// TwinCAT 3 PLC project PLC
// ProgramVersion: 3.1.4023.0
// libraries:
//   Tc2_Standard, * (Beckhoff Automation GmbH)
//   Tc2_System, * (Beckhoff Automation GmbH)
//   Tc3_Module, * (Beckhoff Automation GmbH)
// project tree:
//   / PlcTask.TcTTO
//   POUs/ MAIN.TcPOU
//   DUTs/IO/PDOs/ InfoData_6F19DB2B.TcDUT, Inputs_CC16D1F4.TcDUT, Outputs_D8BAB3B3.TcDUT, WcState_9091E0EB.TcDUT, InfoData_90184F0C.TcDUT, Channel_954C2EED.TcDUT, Channel_60E28ED2.TcDUT, Channel_7DE26195.TcDUT, Channel_2E0D480D.TcDUT, Channel_61FC1536.TcDUT, Channel_16463F74.TcDUT, Channel_707BD1FE.TcDUT, Channel_7D202F58.TcDUT, Channel_6CC0E226.TcDUT, Channel_0F0CD940.TcDUT, Channel_87C95E76.TcDUT, Channel_65B76600.TcDUT, Channel_72DF6336.TcDUT, Channel_22DCD695.TcDUT, Channel_3C1A6500.TcDUT, Channel_B5275D8E.TcDUT, Channel_03CEAA5E.TcDUT, Channel_70C997F3.TcDUT, Channel_1D6668A9.TcDUT, Channel_6B723A16.TcDUT, Channel_460B8C40.TcDUT, Channel_DCF170BB.TcDUT, Channel_26FC8FD8.TcDUT, Channel_FEA3DBF8.TcDUT, Channel_0D1929F0.TcDUT, Channel_6576A681.TcDUT, Channel_2589C8DC.TcDUT, Channel_BF3661CD.TcDUT, Channel_2EC3E8CA.TcDUT, Channel_F5DB8AD1.TcDUT, Channel_6D8B740B.TcDUT, Channel_2DA3FF3C.TcDUT, Channel_0514A8FA.TcDUT, Channel_4E9D1E2D.TcDUT, Channel_78571FB4.TcDUT, Channel_87905831.TcDUT, Channel_099BCCDA.TcDUT, Channel_82ADD076.TcDUT, Channel_332F026B.TcDUT, Channel_A6A8AB45.TcDUT, Channel_A42BCA5C.TcDUT, Channel_08506BCE.TcDUT, Channel_08533804.TcDUT, Channel_A04AC4BD.TcDUT, Channel_77910383.TcDUT, Channel_9BC0092E.TcDUT, Channel_7606D989.TcDUT, Channel_6931CC5B.TcDUT, Channel_F7FDEFA0.TcDUT, Channel_A1C14FB4.TcDUT, Channel_A4B48F2D.TcDUT, Channel_9E293686.TcDUT, Channel_F84AC14F.TcDUT, Channel_2F314509.TcDUT, Channel_D9D48807.TcDUT, Channel_D13646E3.TcDUT, Channel_3263D8D5.TcDUT, Channel_D490E973.TcDUT, KL_6576A681.TcDUT, Channel_64AAC8C7.TcDUT, Channel_471FAA5C.TcDUT, Diag_1F4F4573.TcDUT, Channel_0029832E.TcDUT, Channel_12652743.TcDUT, InfoData_E68C61CD.TcDUT, WcState_0B2B16F9.TcDUT, InfoData_2A97D6CF.TcDUT, Inputs_25A0042B.TcDUT, Outputs_2397A10E.TcDUT
//   DUTs/IO/Boxes/ EK1100_1FC0878B.TcDUT, BK1250_A2FCADE7.TcDUT, KL_5E2F016F.TcDUT, KL_2EA97E3E.TcDUT, KL_1187B721.TcDUT, KL_E991A364.TcDUT, KL_063F0990.TcDUT, KL_5AE00A1C.TcDUT, KL_CFA8830D.TcDUT, KL_DBC0B844.TcDUT, KL_6930B3B2.TcDUT, KL_4F0DAD84.TcDUT, KL_2227C35B.TcDUT, KL1002_BB38DA8F.TcDUT, KL_E653A8C1.TcDUT, KL1012_BB38DA8F.TcDUT, KL1032_BB38DA8F.TcDUT, KL1052_BB38DA8F.TcDUT, KL1104_4A257D2B.TcDUT, KL1114_4A257D2B.TcDUT, KL1124_4A257D2B.TcDUT, KL1154_4A257D2B.TcDUT, KL1164_4A257D2B.TcDUT, KL1184_4A257D2B.TcDUT, KL1194_4A257D2B.TcDUT, KL1212_EC84F46C.TcDUT, KL1232_BB38DA8F.TcDUT, KL1302_BB38DA8F.TcDUT, KL1304_4A257D2B.TcDUT, KL1312_BB38DA8F.TcDUT, KL1314_4A257D2B.TcDUT, KL1352_B54AC54D.TcDUT, KL1362_B54AC54D.TcDUT, KL1382_B54AC54D.TcDUT, KL1402_BB38DA8F.TcDUT, KL1404_4A257D2B.TcDUT, KL1408_8EF4D3E9.TcDUT, KL1412_BB38DA8F.TcDUT, KL1414_4A257D2B.TcDUT, KL1418_8EF4D3E9.TcDUT, KL1434_4A257D2B.TcDUT, KL1488_8EF4D3E9.TcDUT, KL1498_8EF4D3E9.TcDUT, KL1501_EE1D4506.TcDUT, KL_62DC61BC.TcDUT, KL1512_78388DBB.TcDUT, KL1702_BB38DA8F.TcDUT, KL1704_4A257D2B.TcDUT, KL1712_BB38DA8F.TcDUT, KL_BB38DA8F.TcDUT, KL1722_BB38DA8F.TcDUT, KL1804_4A257D2B.TcDUT, KL1808_8EF4D3E9.TcDUT, KL1809_65B88BEE.TcDUT, KL1814_4A257D2B.TcDUT, KL1819_65B88BEE.TcDUT, KL1859_C5B2A062.TcDUT, KL1862_65B88BEE.TcDUT, KL_65B88BEE.TcDUT, KL1872_65B88BEE.TcDUT, KL1889_65B88BEE.TcDUT, KL1904_7F0D69A9.TcDUT, KL1908_7F0D69A9.TcDUT, KL_ABE34026.TcDUT, KL_E882B8F1.TcDUT, KL_52751275.TcDUT, KL2012_DCA75612.TcDUT, KL2022_DCA75612.TcDUT, KL2032_DCA75612.TcDUT, KL2114_E49EE1EF.TcDUT, KL2124_E49EE1EF.TcDUT, KL2134_E49EE1EF.TcDUT, KL2184_E49EE1EF.TcDUT, KL2212_BA18203A.TcDUT, KL1202_EC84F46C.TcDUT, KL2404_E49EE1EF.TcDUT, KL2408_CBAD53BF.TcDUT, KL2424_E49EE1EF.TcDUT, KL2442_DCA75612.TcDUT, KL2488_CBAD53BF.TcDUT, KL2284_008A18FD.TcDUT, KL2502_78388DBB.TcDUT, KL2512_78388DBB.TcDUT, KL2521_D5F34107.TcDUT, KL2531_D5AE5504.TcDUT, KL_5C335388.TcDUT, KL2532_B0461874.TcDUT, KL2535_B0461874.TcDUT, KL_501418F2.TcDUT, KL2541_D5AE5504.TcDUT, KL2542_B0461874.TcDUT, KL2545_B0461874.TcDUT, KL2552_B0461874.TcDUT, KL2602_DCA75612.TcDUT, KL_DCA75612.TcDUT, KL2612_DCA75612.TcDUT, KL2622_DCA75612.TcDUT, KL2631_DE78D366.TcDUT, KL2634_E49EE1EF.TcDUT, KL2641_8487B205.TcDUT, KL_AF699C3C.TcDUT, KL2652_DCA75612.TcDUT, KL_6148C904.TcDUT, KL2701_DE78D366.TcDUT, KL2702_DCA75612.TcDUT, KL2712_DCA75612.TcDUT, KL2722_DCA75612.TcDUT, KL2732_DCA75612.TcDUT, KL2744_E49EE1EF.TcDUT, KL2751_6148C904.TcDUT, KL2761_6148C904.TcDUT, KL2784_E49EE1EF.TcDUT, KL2791_6148C904.TcDUT, KL2794_E49EE1EF.TcDUT, KL2798_CBAD53BF.TcDUT, KL2808_CBAD53BF.TcDUT, KL2819_28D63841.TcDUT, KL2828_CBAD53BF.TcDUT, KL2809_F0D0C9F8.TcDUT, KL2872_F0D0C9F8.TcDUT, KL2889_F0D0C9F8.TcDUT, KL2904_7F0D69A9.TcDUT, KL_F0D0C9F8.TcDUT, KL_CF002DCA.TcDUT, KL_F7A5EEBF.TcDUT, KL_E49EE1EF.TcDUT, KL_F206FFFF.TcDUT, KL_13ED1AE5.TcDUT, KL2774_6148C904.TcDUT, KL_CBAD53BF.TcDUT, KL3001_6148C904.TcDUT, KL3002_B0461874.TcDUT, KL3011_6148C904.TcDUT, KL3012_B0461874.TcDUT, KL3021_6148C904.TcDUT, KL3022_B0461874.TcDUT, KL3041_6148C904.TcDUT, KL3042_B0461874.TcDUT, KL3044_8BE38B75.TcDUT, KL_ACD69469.TcDUT, KL3051_6148C904.TcDUT, KL3052_B0461874.TcDUT, KL3054_8BE38B75.TcDUT, KL3061_6148C904.TcDUT, KL3062_B0461874.TcDUT, KL3064_8BE38B75.TcDUT, KL3102_B0461874.TcDUT, KL3112_B0461874.TcDUT, KL3122_B0461874.TcDUT, KL3132_B0461874.TcDUT, KL3142_78388DBB.TcDUT, KL3152_78388DBB.TcDUT, KL3158_8BE38B75.TcDUT, KL3162_78388DBB.TcDUT, KL3172_78388DBB.TcDUT, KL_78388DBB.TcDUT, KL3182_B0461874.TcDUT, KL3201_6148C904.TcDUT, KL3202_B0461874.TcDUT, KL3204_8BE38B75.TcDUT, KL_8BE38B75.TcDUT, KL3214_8BE38B75.TcDUT, KL3222_B0461874.TcDUT, KL3224_8BE38B75.TcDUT, KL3228_8BE38B75.TcDUT, KL3302_B0461874.TcDUT, KL3311_6148C904.TcDUT, KL3312_B0461874.TcDUT, KL3314_8BE38B75.TcDUT, KL3351_33637CB0.TcDUT, KL_C7B8B3CA.TcDUT, KL3356_E004D4E2.TcDUT, KL_EE1D4506.TcDUT, KL3361_73CB82BA.TcDUT, KL_73CB82BA.TcDUT, KL3362_E98BF8F1.TcDUT, KL6211_60136EA1.TcDUT, KL_9AE543B6.TcDUT, KL_FC0201B8.TcDUT, KL_498D8863.TcDUT, KL_71341691.TcDUT, KL_2B11657C.TcDUT, KL6224_C0F107BD.TcDUT, KL_FC1E3393.TcDUT, KL_C51B1CB0.TcDUT, KL_7EC2CD64.TcDUT, KL_3829421A.TcDUT, KL_9116C2C1.TcDUT, KL6551_528AE398.TcDUT, KL_3325E583.TcDUT, KL_528AE398.TcDUT, KL6781_BE595CA2.TcDUT, KL6811_6148C904.TcDUT, KL6821_F77C82D2.TcDUT, KL6831_BE595CA2.TcDUT, KL6841_BE595CA2.TcDUT, KL6904_B938D612.TcDUT, KL_921B772D.TcDUT, KL_779990DF.TcDUT, KL8001_7761653A.TcDUT, KL8519_8C34650F.TcDUT, KL8524_A4B9216E.TcDUT, KL8528_73A97EC1.TcDUT, KL8548_23451728.TcDUT, KL8610_C571D068.TcDUT, KL_5A83E84C.TcDUT, KL_BF4AA06C.TcDUT, KL_7485E925.TcDUT, KL_372C6BEC.TcDUT, KL_2E5CD6C8.TcDUT, KL_68BDE1E9.TcDUT, KL_84AAE8B6.TcDUT, KL9110_8BEE55F2.TcDUT, KL9160_8BEE55F2.TcDUT, KL9191_962A24DF.TcDUT, KL9210_8BEE55F2.TcDUT, KL9260_8BEE55F2.TcDUT, KL_E4BD2B38.TcDUT, KL9528_8C984603.TcDUT, KL9999_7A10A7F6.TcDUT
//   DUTs/IO/Devices/ SyncUnitTask_2D604ED5.TcDUT, SyncUnitTasks_6FEB8257.TcDUT, SyncUnits_99E584AF.TcDUT
//   DUTs/IO/Topology/ TcTerminals210_1BK1250_A7ABB5AA.TcDUT, TcTerminals210_1EK1100_5C778379.TcDUT, TcTerminals210_2BK1250_CEF74155.TcDUT, TcTerminals210_2EK1100_50C14331.TcDUT, EtherCAT_Master_KL_4053F38C.TcDUT, EtherCAT_Master_KL_8A657514.TcDUT, EtherCAT_Master_KL_B156B97E.TcDUT
//   DUTs/IO/Base/ EtcSlaveBase_82538BE2.TcDUT, EtcSlaveBase_82538BE2.TcDUT, EtcSlaveBase_82538BE2.TcDUT, EtcSlaveTerminalBase_947E5A46.TcDUT, EtcSlaveBoxBase_77A0E4A7.TcDUT, EtcSlaveEndTerminalBase_866C7F0C.TcDUT, InputBase_8311D824.TcDUT, OutputBase_10CEE7DE.TcDUT, EtcMasterBase_62654B43.TcDUT
//   GVLs/ GVL_iXlinker.TcGVL

CONFIGURATION PLC
    RESOURCE PLC ON TwinCAT3
        TASK PlcTask(INTERVAL := T#10ms, PRIORITY := 20);
        PROGRAM MAIN WITH PlcTask : MAIN;
    END_RESOURCE
END_CONFIGURATION

// ---- DUTs/IO/PDOs/InfoData_6F19DB2B.TcDUT
{attribute 'GeneratedUsingTerminal: EK1100-0000-0018'}
{attribute addProperty BoxType "EK1100-0000-0018"}
{attribute addProperty Id "StateAT %I*UINT2"}
{attribute addProperty CRC "1863965483"}
{attribute addProperty Size "2"}
TYPE InfoData_6F19DB2B :
STRUCT
	{attribute addProperty Name "State"}
	State AT %I* : UINT;
END_STRUCT
END_TYPE

// ---- DUTs/IO/PDOs/Inputs_CC16D1F4.TcDUT
{attribute 'GeneratedUsingTerminal: BK1250-0000-0019'}
{attribute addProperty BoxType "BK1250-0000-0019"}
{attribute addProperty Id "CouplerStateAT %I*UINT0"}
{attribute addProperty CRC "3424047604"}
{attribute addProperty Size "0"}
TYPE Inputs_CC16D1F4 EXTENDS InputBase_8311D824 :
STRUCT
	{attribute addProperty Name "CouplerState"}
	CouplerState AT %I* : UINT;
END_STRUCT
END_TYPE

// ---- DUTs/IO/PDOs/Outputs_D8BAB3B3.TcDUT
{attribute 'GeneratedUsingTerminal: BK1250-0000-0019'}
{attribute addProperty BoxType "BK1250-0000-0019"}
{attribute addProperty Id "CouplerCtrlAT %I*UINT0"}
{attribute addProperty CRC "3636114355"}
{attribute addProperty Size "0"}
TYPE Outputs_D8BAB3B3 EXTENDS InputBase_8311D824 :
STRUCT
	{attribute addProperty Name "CouplerCtrl"}
	CouplerCtrl AT %I* : UINT;
END_STRUCT
END_TYPE

// ---- DUTs/IO/PDOs/WcState_9091E0EB.TcDUT
{attribute 'GeneratedUsingTerminal: BK1250-0000-0019'}
{attribute addProperty BoxType "BK1250-0000-0019"}
{attribute addProperty Id "WcStateAT %I*BOOL1InputToggleAT %I*BOOL1"}
{attribute addProperty CRC "2425479403"}
{attribute addProperty Size "2"}
TYPE WcState_9091E0EB :
STRUCT
	{attribute addProperty Name "WcState"}
	WcState AT %I* : BOOL;
	{attribute addProperty Name "InputToggle"}
	InputToggle AT %I* : BOOL;
END_STRUCT
END_TYPE

// ---- DUTs/IO/PDOs/InfoData_90184F0C.TcDUT
{attribute 'GeneratedUsingTerminal: BK1250-0000-0019'}
{attribute addProperty BoxType "BK1250-0000-0019"}
{attribute addProperty Id "AdsAddrAT %I*AMSADDR8AoeNetIdAT %I*AMSNETID6StateAT %I*UINT2"}
{attribute addProperty CRC "2417512204"}
{attribute addProperty Size "16"}
TYPE InfoData_90184F0C EXTENDS InputBase_8311D824 :
STRUCT
	{attribute addProperty Name "AdsAddr"}
	AdsAddr AT %I* : AMSADDR;
	{attribute addProperty Name "AoeNetId"}
	AoeNetId AT %I* : AMSNETID;
	{attribute addProperty Name "State"}
	State AT %I* : UINT;
END_STRUCT
END_TYPE

// ---- DUTs/IO/PDOs/Channel_954C2EED.TcDUT
{attribute 'GeneratedUsingTerminal: KL9940-0050'}
{attribute addProperty BoxType "KL9940-0050"}
{attribute addProperty Id "Key_1AT %I*BOOL0Key_2AT %I*BOOL0Key_3AT %I*BOOL0Key_4AT %I*BOOL0Key_5AT %I*BOOL0Key_6AT %I*BOOL0Key_7AT %I*BOOL0Key_8AT %I*BOOL0Key_9AT %I*BOOL0Key_10AT %I*BOOL0Key_11AT %I*BOOL0Key_12AT %I*BOOL0Key_13AT %I*BOOL0Key_14AT %I*BOOL0Key_15AT %I*BOOL0Key_16AT %I*BOOL0Key_17AT %I*BOOL0Key_18AT %I*BOOL0Key_19AT %I*BOOL0Key_20AT %I*BOOL0Key_21AT %I*BOOL0Key_22AT %I*BOOL0Key_23AT %I*BOOL0Key_24AT %I*BOOL0Key_25AT %I*BOOL0Key_26AT %I*BOOL0Key_27AT %I*BOOL0Key_28AT %I*BOOL0Key_29AT %I*BOOL0Key_30AT %I*BOOL0Key_31AT %I*BOOL0Key_32AT %I*BOOL0Key_33AT %I*BOOL0Key_34AT %I*BOOL0Key_35AT %I*BOOL0Key_36AT %I*BOOL0Key_37AT %I*BOOL0Key_38AT %I*BOOL0Key_39AT %I*BOOL0Key_40AT %I*BOOL0"}
{attribute addProperty CRC "2504797933"}
{attribute addProperty Size "0"}
TYPE Channel_954C2EED EXTENDS InputBase_8311D824 :
STRUCT
	{attribute addProperty Name "Key_1"}
	Key_1 AT %I* : BOOL;
	{attribute addProperty Name "Key_2"}
	Key_2 AT %I* : BOOL;
	{attribute addProperty Name "Key_3"}
	Key_3 AT %I* : BOOL;
	{attribute addProperty Name "Key_4"}
	Key_4 AT %I* : BOOL;
	{attribute addProperty Name "Key_5"}
	Key_5 AT %I* : BOOL;
	{attribute addProperty Name "Key_6"}
	Key_6 AT %I* : BOOL;
	{attribute addProperty Name "Key_7"}
	Key_7 AT %I* : BOOL;
	{attribute addProperty Name "Key_8"}
	Key_8 AT %I* : BOOL;
	{attribute addProperty Name "Key_9"}
	Key_9 AT %I* : BOOL;
	{attribute addProperty Name "Key_10"}
	Key_10 AT %I* : BOOL;
	{attribute addProperty Name "Key_11"}
	Key_11 AT %I* : BOOL;
	{attribute addProperty Name "Key_12"}
	Key_12 AT %I* : BOOL;
	{attribute addProperty Name "Key_13"}
	Key_13 AT %I* : BOOL;
	{attribute addProperty Name "Key_14"}
	Key_14 AT %I* : BOOL;
	{attribute addProperty Name "Key_15"}
	Key_15 AT %I* : BOOL;
	{attribute addProperty Name "Key_16"}
	Key_16 AT %I* : BOOL;
	{attribute addProperty Name "Key_17"}
	Key_17 AT %I* : BOOL;
	{attribute addProperty Name "Key_18"}
	Key_18 AT %I* : BOOL;
	{attribute addProperty Name "Key_19"}
	Key_19 AT %I* : BOOL;
	{attribute addProperty Name "Key_20"}
	Key_20 AT %I* : BOOL;
	{attribute addProperty Name "Key_21"}
	Key_21 AT %I* : BOOL;
	{attribute addProperty Name "Key_22"}
	Key_22 AT %I* : BOOL;
	{attribute addProperty Name "Key_23"}
	Key_23 AT %I* : BOOL;
	{attribute addProperty Name "Key_24"}
	Key_24 AT %I* : BOOL;
	{attribute addProperty Name "Key_25"}
	Key_25 AT %I* : BOOL;
	{attribute addProperty Name "Key_26"}
	Key_26 AT %I* : BOOL;
	{attribute addProperty Name "Key_27"}
	Key_27 AT %I* : BOOL;
	{attribute addProperty Name "Key_28"}
	Key_28 AT %I* : BOOL;
	{attribute addProperty Name "Key_29"}
	Key_29 AT %I* : BOOL;
	{attribute addProperty Name "Key_30"}
	Key_30 AT %I* : BOOL;
	{attribute addProperty Name "Key_31"}
	Key_31 AT %I* : BOOL;
	{attribute addProperty Name "Key_32"}
	Key_32 AT %I* : BOOL;
	{attribute addProperty Name "Key_33"}
	Key_33 AT %I* : BOOL;
	{attribute addProperty Name "Key_34"}
	Key_34 AT %I* : BOOL;
	{attribute addProperty Name "Key_35"}
	Key_35 AT %I* : BOOL;
	{attribute addProperty Name "Key_36"}
	Key_36 AT %I* : BOOL;
	{attribute addProperty Name "Key_37"}
	Key_37 AT %I* : BOOL;
	{attribute addProperty Name "Key_38"}
	Key_38 AT %I* : BOOL;
	{attribute addProperty Name "Key_39"}
	Key_39 AT %I* : BOOL;
	{attribute addProperty Name "Key_40"}
	Key_40 AT %I* : BOOL;
END_STRUCT
END_TYPE

// ---- DUTs/IO/PDOs/Channel_60E28ED2.TcDUT
{attribute 'GeneratedUsingTerminal: KL9900-0054'}
{attribute addProperty BoxType "KL9900-0054"}
{attribute addProperty Id "Key_1AT %I*BOOL0Key_2AT %I*BOOL0Key_3AT %I*BOOL0Key_4AT %I*BOOL0LED_1AT %Q*BOOL0LED_2AT %Q*BOOL0LED_3AT %Q*BOOL0LED_4AT %Q*BOOL0"}
{attribute addProperty CRC "1625460434"}
{attribute addProperty Size "0"}
TYPE Channel_60E28ED2 :
STRUCT
	{attribute addProperty Name "Key_1"}
	Key_1 AT %I* : BOOL;
	{attribute addProperty Name "Key_2"}
	Key_2 AT %I* : BOOL;
	{attribute addProperty Name "Key_3"}
	Key_3 AT %I* : BOOL;
	{attribute addProperty Name "Key_4"}
	Key_4 AT %I* : BOOL;
	{attribute addProperty Name "LED_1"}
	LED_1 AT %Q* : BOOL;
	{attribute addProperty Name "LED_2"}
	LED_2 AT %Q* : BOOL;
	{attribute addProperty Name "LED_3"}
	LED_3 AT %Q* : BOOL;
	{attribute addProperty Name "LED_4"}
	LED_4 AT %Q* : BOOL;
END_STRUCT
END_TYPE

// ---- DUTs/IO/PDOs/Channel_7DE26195.TcDUT
{attribute 'GeneratedUsingTerminal: KL9900-0055'}
{attribute addProperty BoxType "KL9900-0055"}
{attribute addProperty Id "Key_1AT %I*BOOL0Key_2AT %I*BOOL0Key_3AT %I*BOOL0Key_4AT %I*BOOL0Key_5AT %I*BOOL0Key_6AT %I*BOOL0Key_7AT %I*BOOL0Key_8AT %I*BOOL0LED_1AT %Q*BOOL0LED_2AT %Q*BOOL0LED_3AT %Q*BOOL0LED_4AT %Q*BOOL0LED_5AT %Q*BOOL0LED_6AT %Q*BOOL0LED_7AT %Q*BOOL0LED_8AT %Q*BOOL0"}
{attribute addProperty CRC "2111988117"}
{attribute addProperty Size "0"}
TYPE Channel_7DE26195 :
STRUCT
	{attribute addProperty Name "Key_1"}
	Key_1 AT %I* : BOOL;
	{attribute addProperty Name "Key_2"}
	Key_2 AT %I* : BOOL;
	{attribute addProperty Name "Key_3"}
	Key_3 AT %I* : BOOL;
	{attribute addProperty Name "Key_4"}
	Key_4 AT %I* : BOOL;
	{attribute addProperty Name "Key_5"}
	Key_5 AT %I* : BOOL;
	{attribute addProperty Name "Key_6"}
	Key_6 AT %I* : BOOL;
	{attribute addProperty Name "Key_7"}
	Key_7 AT %I* : BOOL;
	{attribute addProperty Name "Key_8"}
	Key_8 AT %I* : BOOL;
	{attribute addProperty Name "LED_1"}
	LED_1 AT %Q* : BOOL;
	{attribute addProperty Name "LED_2"}
	LED_2 AT %Q* : BOOL;
	{attribute addProperty Name "LED_3"}
	LED_3 AT %Q* : BOOL;
	{attribute addProperty Name "LED_4"}
	LED_4 AT %Q* : BOOL;
	{attribute addProperty Name "LED_5"}
	LED_5 AT %Q* : BOOL;
	{attribute addProperty Name "LED_6"}
	LED_6 AT %Q* : BOOL;
	{attribute addProperty Name "LED_7"}
	LED_7 AT %Q* : BOOL;
	{attribute addProperty Name "LED_8"}
	LED_8 AT %Q* : BOOL;
END_STRUCT
END_TYPE

// ---- DUTs/IO/PDOs/Channel_2E0D480D.TcDUT
{attribute 'GeneratedUsingTerminal: KL9900-0056'}
{attribute addProperty BoxType "KL9900-0056"}
{attribute addProperty Id "Key_1AT %I*BOOL0Key_2AT %I*BOOL0Key_3AT %I*BOOL0Key_4AT %I*BOOL0Key_5AT %I*BOOL0Key_6AT %I*BOOL0Key_7AT %I*BOOL0Key_8AT %I*BOOL0Key_9AT %I*BOOL0Key_10AT %I*BOOL0Key_11AT %I*BOOL0Key_12AT %I*BOOL0LED_1AT %Q*BOOL0LED_2AT %Q*BOOL0LED_3AT %Q*BOOL0LED_4AT %Q*BOOL0LED_5AT %Q*BOOL0LED_6AT %Q*BOOL0LED_7AT %Q*BOOL0LED_8AT %Q*BOOL0LED_9AT %Q*BOOL0LED_10AT %Q*BOOL0LED_11AT %Q*BOOL0LED_12AT %Q*BOOL0"}
{attribute addProperty CRC "772622349"}
{attribute addProperty Size "0"}
TYPE Channel_2E0D480D :
STRUCT
	{attribute addProperty Name "Key_1"}
	Key_1 AT %I* : BOOL;
	{attribute addProperty Name "Key_2"}
	Key_2 AT %I* : BOOL;
	{attribute addProperty Name "Key_3"}
	Key_3 AT %I* : BOOL;
	{attribute addProperty Name "Key_4"}
	Key_4 AT %I* : BOOL;
	{attribute addProperty Name "Key_5"}
	Key_5 AT %I* : BOOL;
	{attribute addProperty Name "Key_6"}
	Key_6 AT %I* : BOOL;
	{attribute addProperty Name "Key_7"}
	Key_7 AT %I* : BOOL;
	{attribute addProperty Name "Key_8"}
	Key_8 AT %I* : BOOL;
	{attribute addProperty Name "Key_9"}
	Key_9 AT %I* : BOOL;
	{attribute addProperty Name "Key_10"}
	Key_10 AT %I* : BOOL;
	{attribute addProperty Name "Key_11"}
	Key_11 AT %I* : BOOL;
	{attribute addProperty Name "Key_12"}
	Key_12 AT %I* : BOOL;
	{attribute addProperty Name "LED_1"}
	LED_1 AT %Q* : BOOL;
	{attribute addProperty Name "LED_2"}
	LED_2 AT %Q* : BOOL;
	{attribute addProperty Name "LED_3"}
	LED_3 AT %Q* : BOOL;
	{attribute addProperty Name "LED_4"}
	LED_4 AT %Q* : BOOL;
	{attribute addProperty Name "LED_5"}
	LED_5 AT %Q* : BOOL;
	{attribute addProperty Name "LED_6"}
	LED_6 AT %Q* : BOOL;
	{attribute addProperty Name "LED_7"}
	LED_7 AT %Q* : BOOL;
	{attribute addProperty Name "LED_8"}
	LED_8 AT %Q* : BOOL;
	{attribute addProperty Name "LED_9"}
	LED_9 AT %Q* : BOOL;
	{attribute addProperty Name "LED_10"}
	LED_10 AT %Q* : BOOL;
	{attribute addProperty Name "LED_11"}
	LED_11 AT %Q* : BOOL;
	{attribute addProperty Name "LED_12"}
	LED_12 AT %Q* : BOOL;
END_STRUCT
END_TYPE

// ---- DUTs/IO/PDOs/Channel_61FC1536.TcDUT
{attribute 'GeneratedUsingTerminal: KL9900-0057'}
{attribute addProperty BoxType "KL9900-0057"}
{attribute addProperty Id "Key_1AT %I*BOOL0Key_2AT %I*BOOL0Key_3AT %I*BOOL0Key_4AT %I*BOOL0Key_5AT %I*BOOL0Key_6AT %I*BOOL0Key_7AT %I*BOOL0Key_8AT %I*BOOL0Key_9AT %I*BOOL0Key_10AT %I*BOOL0Key_11AT %I*BOOL0Key_12AT %I*BOOL0Key_13AT %I*BOOL0Key_14AT %I*BOOL0Key_15AT %I*BOOL0Key_16AT %I*BOOL0LED_1AT %Q*BOOL0LED_2AT %Q*BOOL0LED_3AT %Q*BOOL0LED_4AT %Q*BOOL0LED_5AT %Q*BOOL0LED_6AT %Q*BOOL0LED_7AT %Q*BOOL0LED_8AT %Q*BOOL0LED_9AT %Q*BOOL0LED_10AT %Q*BOOL0LED_11AT %Q*BOOL0LED_12AT %Q*BOOL0LED_13AT %Q*BOOL0LED_14AT %Q*BOOL0LED_15AT %Q*BOOL0LED_16AT %Q*BOOL0"}
{attribute addProperty CRC "1643910454"}
{attribute addProperty Size "0"}
TYPE Channel_61FC1536 :
STRUCT
	{attribute addProperty Name "Key_1"}
	Key_1 AT %I* : BOOL;
	{attribute addProperty Name "Key_2"}
	Key_2 AT %I* : BOOL;
	{attribute addProperty Name "Key_3"}
	Key_3 AT %I* : BOOL;
	{attribute addProperty Name "Key_4"}
	Key_4 AT %I* : BOOL;
	{attribute addProperty Name "Key_5"}
	Key_5 AT %I* : BOOL;
	{attribute addProperty Name "Key_6"}
	Key_6 AT %I* : BOOL;
	{attribute addProperty Name "Key_7"}
	Key_7 AT %I* : BOOL;
	{attribute addProperty Name "Key_8"}
	Key_8 AT %I* : BOOL;
	{attribute addProperty Name "Key_9"}
	Key_9 AT %I* : BOOL;
	{attribute addProperty Name "Key_10"}
	Key_10 AT %I* : BOOL;
	{attribute addProperty Name "Key_11"}
	Key_11 AT %I* : BOOL;
	{attribute addProperty Name "Key_12"}
	Key_12 AT %I* : BOOL;
	{attribute addProperty Name "Key_13"}
	Key_13 AT %I* : BOOL;
	{attribute addProperty Name "Key_14"}
	Key_14 AT %I* : BOOL;
	{attribute addProperty Name "Key_15"}
	Key_15 AT %I* : BOOL;
	{attribute addProperty Name "Key_16"}
	Key_16 AT %I* : BOOL;
	{attribute addProperty Name "LED_1"}
	LED_1 AT %Q* : BOOL;
	{attribute addProperty Name "LED_2"}
	LED_2 AT %Q* : BOOL;
	{attribute addProperty Name "LED_3"}
	LED_3 AT %Q* : BOOL;
	{attribute addProperty Name "LED_4"}
	LED_4 AT %Q* : BOOL;
	{attribute addProperty Name "LED_5"}
	LED_5 AT %Q* : BOOL;
	{attribute addProperty Name "LED_6"}
	LED_6 AT %Q* : BOOL;
	{attribute addProperty Name "LED_7"}
	LED_7 AT %Q* : BOOL;
	{attribute addProperty Name "LED_8"}
	LED_8 AT %Q* : BOOL;
	{attribute addProperty Name "LED_9"}
	LED_9 AT %Q* : BOOL;
	{attribute addProperty Name "LED_10"}
	LED_10 AT %Q* : BOOL;
	{attribute addProperty Name "LED_11"}
	LED_11 AT %Q* : BOOL;
	{attribute addProperty Name "LED_12"}
	LED_12 AT %Q* : BOOL;
	{attribute addProperty Name "LED_13"}
	LED_13 AT %Q* : BOOL;
	{attribute addProperty Name "LED_14"}
	LED_14 AT %Q* : BOOL;
	{attribute addProperty Name "LED_15"}
	LED_15 AT %Q* : BOOL;
	{attribute addProperty Name "LED_16"}
	LED_16 AT %Q* : BOOL;
END_STRUCT
END_TYPE

// ---- DUTs/IO/PDOs/Channel_16463F74.TcDUT
{attribute 'GeneratedUsingTerminal: KL9900-0058'}
{attribute addProperty BoxType "KL9900-0058"}
{attribute addProperty Id "Key_1AT %I*BOOL0Key_2AT %I*BOOL0Key_3AT %I*BOOL0Key_4AT %I*BOOL0Key_5AT %I*BOOL0Key_6AT %I*BOOL0Key_7AT %I*BOOL0Key_8AT %I*BOOL0Key_9AT %I*BOOL0Key_10AT %I*BOOL0Key_11AT %I*BOOL0Key_12AT %I*BOOL0Key_13AT %I*BOOL0Key_14AT %I*BOOL0Key_15AT %I*BOOL0Key_16AT %I*BOOL0Key_17AT %I*BOOL0Key_18AT %I*BOOL0Key_19AT %I*BOOL0Key_20AT %I*BOOL0LED_1AT %Q*BOOL0LED_2AT %Q*BOOL0LED_3AT %Q*BOOL0LED_4AT %Q*BOOL0LED_5AT %Q*BOOL0LED_6AT %Q*BOOL0LED_7AT %Q*BOOL0LED_8AT %Q*BOOL0LED_9AT %Q*BOOL0LED_10AT %Q*BOOL0LED_11AT %Q*BOOL0LED_12AT %Q*BOOL0LED_13AT %Q*BOOL0LED_14AT %Q*BOOL0LED_15AT %Q*BOOL0LED_16AT %Q*BOOL0LED_17AT %Q*BOOL0LED_18AT %Q*BOOL0LED_19AT %Q*BOOL0LED_20AT %Q*BOOL0"}
{attribute addProperty CRC "373702516"}
{attribute addProperty Size "0"}
TYPE Channel_16463F74 :
STRUCT
	{attribute addProperty Name "Key_1"}
	Key_1 AT %I* : BOOL;
	{attribute addProperty Name "Key_2"}
	Key_2 AT %I* : BOOL;
	{attribute addProperty Name "Key_3"}
	Key_3 AT %I* : BOOL;
	{attribute addProperty Name "Key_4"}
	Key_4 AT %I* : BOOL;
	{attribute addProperty Name "Key_5"}
	Key_5 AT %I* : BOOL;
	{attribute addProperty Name "Key_6"}
	Key_6 AT %I* : BOOL;
	{attribute addProperty Name "Key_7"}
	Key_7 AT %I* : BOOL;
	{attribute addProperty Name "Key_8"}
	Key_8 AT %I* : BOOL;
	{attribute addProperty Name "Key_9"}
	Key_9 AT %I* : BOOL;
	{attribute addProperty Name "Key_10"}
	Key_10 AT %I* : BOOL;
	{attribute addProperty Name "Key_11"}
	Key_11 AT %I* : BOOL;
	{attribute addProperty Name "Key_12"}
	Key_12 AT %I* : BOOL;
	{attribute addProperty Name "Key_13"}
	Key_13 AT %I* : BOOL;
	{attribute addProperty Name "Key_14"}
	Key_14 AT %I* : BOOL;
	{attribute addProperty Name "Key_15"}
	Key_15 AT %I* : BOOL;
	{attribute addProperty Name "Key_16"}
	Key_16 AT %I* : BOOL;
	{attribute addProperty Name "Key_17"}
	Key_17 AT %I* : BOOL;
	{attribute addProperty Name "Key_18"}
	Key_18 AT %I* : BOOL;
	{attribute addProperty Name "Key_19"}
	Key_19 AT %I* : BOOL;
	{attribute addProperty Name "Key_20"}
	Key_20 AT %I* : BOOL;
	{attribute addProperty Name "LED_1"}
	LED_1 AT %Q* : BOOL;
	{attribute addProperty Name "LED_2"}
	LED_2 AT %Q* : BOOL;
	{attribute addProperty Name "LED_3"}
	LED_3 AT %Q* : BOOL;
	{attribute addProperty Name "LED_4"}
	LED_4 AT %Q* : BOOL;
	{attribute addProperty Name "LED_5"}
	LED_5 AT %Q* : BOOL;
	{attribute addProperty Name "LED_6"}
	LED_6 AT %Q* : BOOL;
	{attribute addProperty Name "LED_7"}
	LED_7 AT %Q* : BOOL;
	{attribute addProperty Name "LED_8"}
	LED_8 AT %Q* : BOOL;
	{attribute addProperty Name "LED_9"}
	LED_9 AT %Q* : BOOL;
	{attribute addProperty Name "LED_10"}
	LED_10 AT %Q* : BOOL;
	{attribute addProperty Name "LED_11"}
	LED_11 AT %Q* : BOOL;
	{attribute addProperty Name "LED_12"}
	LED_12 AT %Q* : BOOL;
	{attribute addProperty Name "LED_13"}
	LED_13 AT %Q* : BOOL;
	{attribute addProperty Name "LED_14"}
	LED_14 AT %Q* : BOOL;
	{attribute addProperty Name "LED_15"}
	LED_15 AT %Q* : BOOL;
	{attribute addProperty Name "LED_16"}
	LED_16 AT %Q* : BOOL;
	{attribute addProperty Name "LED_17"}
	LED_17 AT %Q* : BOOL;
	{attribute addProperty Name "LED_18"}
	LED_18 AT %Q* : BOOL;
	{attribute addProperty Name "LED_19"}
	LED_19 AT %Q* : BOOL;
	{attribute addProperty Name "LED_20"}
	LED_20 AT %Q* : BOOL;
END_STRUCT
END_TYPE

// ---- DUTs/IO/PDOs/Channel_707BD1FE.TcDUT
{attribute 'GeneratedUsingTerminal: KL9900-0059'}
{attribute addProperty BoxType "KL9900-0059"}
{attribute addProperty Id "Key_1AT %I*BOOL0Key_2AT %I*BOOL0Key_3AT %I*BOOL0Key_4AT %I*BOOL0Key_5AT %I*BOOL0Key_6AT %I*BOOL0Key_7AT %I*BOOL0Key_8AT %I*BOOL0Key_9AT %I*BOOL0Key_10AT %I*BOOL0Key_11AT %I*BOOL0Key_12AT %I*BOOL0Key_13AT %I*BOOL0Key_14AT %I*BOOL0Key_15AT %I*BOOL0Key_16AT %I*BOOL0Key_17AT %I*BOOL0Key_18AT %I*BOOL0Key_19AT %I*BOOL0Key_20AT %I*BOOL0Key_21AT %I*BOOL0Key_22AT %I*BOOL0Key_23AT %I*BOOL0Key_24AT %I*BOOL0LED_1AT %Q*BOOL0LED_2AT %Q*BOOL0LED_3AT %Q*BOOL0LED_4AT %Q*BOOL0LED_5AT %Q*BOOL0LED_6AT %Q*BOOL0LED_7AT %Q*BOOL0LED_8AT %Q*BOOL0LED_9AT %Q*BOOL0LED_10AT %Q*BOOL0LED_11AT %Q*BOOL0LED_12AT %Q*BOOL0LED_13AT %Q*BOOL0LED_14AT %Q*BOOL0LED_15AT %Q*BOOL0LED_16AT %Q*BOOL0LED_17AT %Q*BOOL0LED_18AT %Q*BOOL0LED_19AT %Q*BOOL0LED_20AT %Q*BOOL0LED_21AT %Q*BOOL0LED_22AT %Q*BOOL0LED_23AT %Q*BOOL0LED_24AT %Q*BOOL0"}
{attribute addProperty CRC "1887162878"}
{attribute addProperty Size "0"}
TYPE Channel_707BD1FE :
STRUCT
	{attribute addProperty Name "Key_1"}
	Key_1 AT %I* : BOOL;
	{attribute addProperty Name "Key_2"}
	Key_2 AT %I* : BOOL;
	{attribute addProperty Name "Key_3"}
	Key_3 AT %I* : BOOL;
	{attribute addProperty Name "Key_4"}
	Key_4 AT %I* : BOOL;
	{attribute addProperty Name "Key_5"}
	Key_5 AT %I* : BOOL;
	{attribute addProperty Name "Key_6"}
	Key_6 AT %I* : BOOL;
	{attribute addProperty Name "Key_7"}
	Key_7 AT %I* : BOOL;
	{attribute addProperty Name "Key_8"}
	Key_8 AT %I* : BOOL;
	{attribute addProperty Name "Key_9"}
	Key_9 AT %I* : BOOL;
	{attribute addProperty Name "Key_10"}
	Key_10 AT %I* : BOOL;
	{attribute addProperty Name "Key_11"}
	Key_11 AT %I* : BOOL;
	{attribute addProperty Name "Key_12"}
	Key_12 AT %I* : BOOL;
	{attribute addProperty Name "Key_13"}
	Key_13 AT %I* : BOOL;
	{attribute addProperty Name "Key_14"}
	Key_14 AT %I* : BOOL;
	{attribute addProperty Name "Key_15"}
	Key_15 AT %I* : BOOL;
	{attribute addProperty Name "Key_16"}
	Key_16 AT %I* : BOOL;
	{attribute addProperty Name "Key_17"}
	Key_17 AT %I* : BOOL;
	{attribute addProperty Name "Key_18"}
	Key_18 AT %I* : BOOL;
	{attribute addProperty Name "Key_19"}
	Key_19 AT %I* : BOOL;
	{attribute addProperty Name "Key_20"}
	Key_20 AT %I* : BOOL;
	{attribute addProperty Name "Key_21"}
	Key_21 AT %I* : BOOL;
	{attribute addProperty Name "Key_22"}
	Key_22 AT %I* : BOOL;
	{attribute addProperty Name "Key_23"}
	Key_23 AT %I* : BOOL;
	{attribute addProperty Name "Key_24"}
	Key_24 AT %I* : BOOL;
	{attribute addProperty Name "LED_1"}
	LED_1 AT %Q* : BOOL;
	{attribute addProperty Name "LED_2"}
	LED_2 AT %Q* : BOOL;
	{attribute addProperty Name "LED_3"}
	LED_3 AT %Q* : BOOL;
	{attribute addProperty Name "LED_4"}
	LED_4 AT %Q* : BOOL;
	{attribute addProperty Name "LED_5"}
	LED_5 AT %Q* : BOOL;
	{attribute addProperty Name "LED_6"}
	LED_6 AT %Q* : BOOL;
	{attribute addProperty Name "LED_7"}
	LED_7 AT %Q* : BOOL;
	{attribute addProperty Name "LED_8"}
	LED_8 AT %Q* : BOOL;
	{attribute addProperty Name "LED_9"}
	LED_9 AT %Q* : BOOL;
	{attribute addProperty Name "LED_10"}
	LED_10 AT %Q* : BOOL;
	{attribute addProperty Name "LED_11"}
	LED_11 AT %Q* : BOOL;
	{attribute addProperty Name "LED_12"}
	LED_12 AT %Q* : BOOL;
	{attribute addProperty Name "LED_13"}
	LED_13 AT %Q* : BOOL;
	{attribute addProperty Name "LED_14"}
	LED_14 AT %Q* : BOOL;
	{attribute addProperty Name "LED_15"}
	LED_15 AT %Q* : BOOL;
	{attribute addProperty Name "LED_16"}
	LED_16 AT %Q* : BOOL;
	{attribute addProperty Name "LED_17"}
	LED_17 AT %Q* : BOOL;
	{attribute addProperty Name "LED_18"}
	LED_18 AT %Q* : BOOL;
	{attribute addProperty Name "LED_19"}
	LED_19 AT %Q* : BOOL;
	{attribute addProperty Name "LED_20"}
	LED_20 AT %Q* : BOOL;
	{attribute addProperty Name "LED_21"}
	LED_21 AT %Q* : BOOL;
	{attribute addProperty Name "LED_22"}
	LED_22 AT %Q* : BOOL;
	{attribute addProperty Name "LED_23"}
	LED_23 AT %Q* : BOOL;
	{attribute addProperty Name "LED_24"}
	LED_24 AT %Q* : BOOL;
END_STRUCT
END_TYPE

// ---- DUTs/IO/PDOs/Channel_7D202F58.TcDUT
{attribute 'GeneratedUsingTerminal: KL9900-0060'}
{attribute addProperty BoxType "KL9900-0060"}
{attribute addProperty Id "Key_1AT %I*BOOL0Key_2AT %I*BOOL0Key_3AT %I*BOOL0Key_4AT %I*BOOL0Key_5AT %I*BOOL0Key_6AT %I*BOOL0Key_7AT %I*BOOL0Key_8AT %I*BOOL0Key_9AT %I*BOOL0Key_10AT %I*BOOL0Key_11AT %I*BOOL0Key_12AT %I*BOOL0Key_13AT %I*BOOL0Key_14AT %I*BOOL0Key_15AT %I*BOOL0Key_16AT %I*BOOL0Key_17AT %I*BOOL0Key_18AT %I*BOOL0Key_19AT %I*BOOL0Key_20AT %I*BOOL0Key_21AT %I*BOOL0Key_22AT %I*BOOL0Key_23AT %I*BOOL0Key_24AT %I*BOOL0Key_25AT %I*BOOL0Key_26AT %I*BOOL0Key_27AT %I*BOOL0Key_28AT %I*BOOL0LED_1AT %Q*BOOL0LED_2AT %Q*BOOL0LED_3AT %Q*BOOL0LED_4AT %Q*BOOL0LED_5AT %Q*BOOL0LED_6AT %Q*BOOL0LED_7AT %Q*BOOL0LED_8AT %Q*BOOL0LED_9AT %Q*BOOL0LED_10AT %Q*BOOL0LED_11AT %Q*BOOL0LED_12AT %Q*BOOL0LED_13AT %Q*BOOL0LED_14AT %Q*BOOL0LED_15AT %Q*BOOL0LED_16AT %Q*BOOL0LED_17AT %Q*BOOL0LED_18AT %Q*BOOL0LED_19AT %Q*BOOL0LED_20AT %Q*BOOL0LED_21AT %Q*BOOL0LED_22AT %Q*BOOL0LED_23AT %Q*BOOL0LED_24AT %Q*BOOL0LED_25AT %Q*BOOL0LED_26AT %Q*BOOL0LED_27AT %Q*BOOL0LED_28AT %Q*BOOL0"}
{attribute addProperty CRC "2099261272"}
{attribute addProperty Size "0"}
TYPE Channel_7D202F58 :
STRUCT
	{attribute addProperty Name "Key_1"}
	Key_1 AT %I* : BOOL;
	{attribute addProperty Name "Key_2"}
	Key_2 AT %I* : BOOL;
	{attribute addProperty Name "Key_3"}
	Key_3 AT %I* : BOOL;
	{attribute addProperty Name "Key_4"}
	Key_4 AT %I* : BOOL;
	{attribute addProperty Name "Key_5"}
	Key_5 AT %I* : BOOL;
	{attribute addProperty Name "Key_6"}
	Key_6 AT %I* : BOOL;
	{attribute addProperty Name "Key_7"}
	Key_7 AT %I* : BOOL;
	{attribute addProperty Name "Key_8"}
	Key_8 AT %I* : BOOL;
	{attribute addProperty Name "Key_9"}
	Key_9 AT %I* : BOOL;
	{attribute addProperty Name "Key_10"}
	Key_10 AT %I* : BOOL;
	{attribute addProperty Name "Key_11"}
	Key_11 AT %I* : BOOL;
	{attribute addProperty Name "Key_12"}
	Key_12 AT %I* : BOOL;
	{attribute addProperty Name "Key_13"}
	Key_13 AT %I* : BOOL;
	{attribute addProperty Name "Key_14"}
	Key_14 AT %I* : BOOL;
	{attribute addProperty Name "Key_15"}
	Key_15 AT %I* : BOOL;
	{attribute addProperty Name "Key_16"}
	Key_16 AT %I* : BOOL;
	{attribute addProperty Name "Key_17"}
	Key_17 AT %I* : BOOL;
	{attribute addProperty Name "Key_18"}
	Key_18 AT %I* : BOOL;
	{attribute addProperty Name "Key_19"}
	Key_19 AT %I* : BOOL;
	{attribute addProperty Name "Key_20"}
	Key_20 AT %I* : BOOL;
	{attribute addProperty Name "Key_21"}
	Key_21 AT %I* : BOOL;
	{attribute addProperty Name "Key_22"}
	Key_22 AT %I* : BOOL;
	{attribute addProperty Name "Key_23"}
	Key_23 AT %I* : BOOL;
	{attribute addProperty Name "Key_24"}
	Key_24 AT %I* : BOOL;
	{attribute addProperty Name "Key_25"}
	Key_25 AT %I* : BOOL;
	{attribute addProperty Name "Key_26"}
	Key_26 AT %I* : BOOL;
	{attribute addProperty Name "Key_27"}
	Key_27 AT %I* : BOOL;
	{attribute addProperty Name "Key_28"}
	Key_28 AT %I* : BOOL;
	{attribute addProperty Name "LED_1"}
	LED_1 AT %Q* : BOOL;
	{attribute addProperty Name "LED_2"}
	LED_2 AT %Q* : BOOL;
	{attribute addProperty Name "LED_3"}
	LED_3 AT %Q* : BOOL;
	{attribute addProperty Name "LED_4"}
	LED_4 AT %Q* : BOOL;
	{attribute addProperty Name "LED_5"}
	LED_5 AT %Q* : BOOL;
	{attribute addProperty Name "LED_6"}
	LED_6 AT %Q* : BOOL;
	{attribute addProperty Name "LED_7"}
	LED_7 AT %Q* : BOOL;
	{attribute addProperty Name "LED_8"}
	LED_8 AT %Q* : BOOL;
	{attribute addProperty Name "LED_9"}
	LED_9 AT %Q* : BOOL;
	{attribute addProperty Name "LED_10"}
	LED_10 AT %Q* : BOOL;
	{attribute addProperty Name "LED_11"}
	LED_11 AT %Q* : BOOL;
	{attribute addProperty Name "LED_12"}
	LED_12 AT %Q* : BOOL;
	{attribute addProperty Name "LED_13"}
	LED_13 AT %Q* : BOOL;
	{attribute addProperty Name "LED_14"}
	LED_14 AT %Q* : BOOL;
	{attribute addProperty Name "LED_15"}
	LED_15 AT %Q* : BOOL;
	{attribute addProperty Name "LED_16"}
	LED_16 AT %Q* : BOOL;
	{attribute addProperty Name "LED_17"}
	LED_17 AT %Q* : BOOL;
	{attribute addProperty Name "LED_18"}
	LED_18 AT %Q* : BOOL;
	{attribute addProperty Name "LED_19"}
	LED_19 AT %Q* : BOOL;
	{attribute addProperty Name "LED_20"}
	LED_20 AT %Q* : BOOL;
	{attribute addProperty Name "LED_21"}
	LED_21 AT %Q* : BOOL;
	{attribute addProperty Name "LED_22"}
	LED_22 AT %Q* : BOOL;
	{attribute addProperty Name "LED_23"}
	LED_23 AT %Q* : BOOL;
	{attribute addProperty Name "LED_24"}
	LED_24 AT %Q* : BOOL;
	{attribute addProperty Name "LED_25"}
	LED_25 AT %Q* : BOOL;
	{attribute addProperty Name "LED_26"}
	LED_26 AT %Q* : BOOL;
	{attribute addProperty Name "LED_27"}
	LED_27 AT %Q* : BOOL;
	{attribute addProperty Name "LED_28"}
	LED_28 AT %Q* : BOOL;
END_STRUCT
END_TYPE

// ---- DUTs/IO/PDOs/Channel_6CC0E226.TcDUT
{attribute 'GeneratedUsingTerminal: KL9900-0063'}
{attribute addProperty BoxType "KL9900-0063"}
{attribute addProperty Id "Key_1AT %I*BOOL0Key_2AT %I*BOOL0Key_3AT %I*BOOL0Input_1AT %I*BOOL0Input_2AT %I*BOOL0Input_3AT %I*BOOL0LED_1AT %Q*BOOL0LED_2AT %Q*BOOL0LED_3AT %Q*BOOL0"}
{attribute addProperty CRC "1824580134"}
{attribute addProperty Size "0"}
TYPE Channel_6CC0E226 :
STRUCT
	{attribute addProperty Name "Key_1"}
	Key_1 AT %I* : BOOL;
	{attribute addProperty Name "Key_2"}
	Key_2 AT %I* : BOOL;
	{attribute addProperty Name "Key_3"}
	Key_3 AT %I* : BOOL;
	{attribute addProperty Name "Input_1"}
	Input_1 AT %I* : BOOL;
	{attribute addProperty Name "Input_2"}
	Input_2 AT %I* : BOOL;
	{attribute addProperty Name "Input_3"}
	Input_3 AT %I* : BOOL;
	{attribute addProperty Name "LED_1"}
	LED_1 AT %Q* : BOOL;
	{attribute addProperty Name "LED_2"}
	LED_2 AT %Q* : BOOL;
	{attribute addProperty Name "LED_3"}
	LED_3 AT %Q* : BOOL;
END_STRUCT
END_TYPE

// ---- DUTs/IO/PDOs/Channel_0F0CD940.TcDUT
{attribute 'GeneratedUsingTerminal: KL9900-0064'}
{attribute addProperty BoxType "KL9900-0064"}
{attribute addProperty Id "Key_1AT %I*BOOL0Key_2AT %I*BOOL0Key_3AT %I*BOOL0Key_4AT %I*BOOL0Input_1AT %I*BOOL0Input_2AT %I*BOOL0Input_3AT %I*BOOL0Input_4AT %I*BOOL0LED_1AT %Q*BOOL0LED_2AT %Q*BOOL0LED_3AT %Q*BOOL0LED_4AT %Q*BOOL0"}
{attribute addProperty CRC "252500288"}
{attribute addProperty Size "0"}
TYPE Channel_0F0CD940 :
STRUCT
	{attribute addProperty Name "Key_1"}
	Key_1 AT %I* : BOOL;
	{attribute addProperty Name "Key_2"}
	Key_2 AT %I* : BOOL;
	{attribute addProperty Name "Key_3"}
	Key_3 AT %I* : BOOL;
	{attribute addProperty Name "Key_4"}
	Key_4 AT %I* : BOOL;
	{attribute addProperty Name "Input_1"}
	Input_1 AT %I* : BOOL;
	{attribute addProperty Name "Input_2"}
	Input_2 AT %I* : BOOL;
	{attribute addProperty Name "Input_3"}
	Input_3 AT %I* : BOOL;
	{attribute addProperty Name "Input_4"}
	Input_4 AT %I* : BOOL;
	{attribute addProperty Name "LED_1"}
	LED_1 AT %Q* : BOOL;
	{attribute addProperty Name "LED_2"}
	LED_2 AT %Q* : BOOL;
	{attribute addProperty Name "LED_3"}
	LED_3 AT %Q* : BOOL;
	{attribute addProperty Name "LED_4"}
	LED_4 AT %Q* : BOOL;
END_STRUCT
END_TYPE

// ---- DUTs/IO/PDOs/Channel_87C95E76.TcDUT
{attribute 'GeneratedUsingTerminal: KL1002'}
{attribute addProperty BoxType "KL1002"}
{attribute addProperty Id "InputAT %I*BOOL0"}
{attribute addProperty CRC "2278121078"}
{attribute addProperty Size "0"}
TYPE Channel_87C95E76 EXTENDS InputBase_8311D824 :
STRUCT
	{attribute addProperty Name "Input"}
	Input AT %I* : BOOL;
END_STRUCT
END_TYPE

// ---- DUTs/IO/PDOs/Channel_65B76600.TcDUT
{attribute 'GeneratedUsingTerminal: KL9900-0062'}
{attribute addProperty BoxType "KL9900-0062"}
{attribute addProperty Id "E_StopAT %I*BOOL0"}
{attribute addProperty CRC "1706518016"}
{attribute addProperty Size "0"}
TYPE Channel_65B76600 EXTENDS InputBase_8311D824 :
STRUCT
	{attribute addProperty Name "E_Stop"}
	E_Stop AT %I* : BOOL;
END_STRUCT
END_TYPE

// ---- DUTs/IO/PDOs/Channel_72DF6336.TcDUT
{attribute 'GeneratedUsingTerminal: KL1212'}
{attribute addProperty BoxType "KL1212"}
{attribute addProperty Id "InputAT %I*BOOL0ErrorAT %I*BOOL0PowerAT %Q*BOOL0"}
{attribute addProperty CRC "1927242550"}
{attribute addProperty Size "0"}
TYPE Channel_72DF6336 :
STRUCT
	{attribute addProperty Name "Input"}
	Input AT %I* : BOOL;
	{attribute addProperty Name "Error"}
	Error AT %I* : BOOL;
	{attribute addProperty Name "Power"}
	Power AT %Q* : BOOL;
END_STRUCT
END_TYPE

// ---- DUTs/IO/PDOs/Channel_22DCD695.TcDUT
{attribute 'GeneratedUsingTerminal: KL1352'}
{attribute addProperty BoxType "KL1352"}
{attribute addProperty Id "InputAT %I*BOOL0ErrorAT %I*BOOL0"}
{attribute addProperty CRC "584898197"}
{attribute addProperty Size "0"}
TYPE Channel_22DCD695 EXTENDS InputBase_8311D824 :
STRUCT
	{attribute addProperty Name "Input"}
	Input AT %I* : BOOL;
	{attribute addProperty Name "Error"}
	Error AT %I* : BOOL;
END_STRUCT
END_TYPE

// ---- DUTs/IO/PDOs/Channel_3C1A6500.TcDUT
{attribute 'GeneratedUsingTerminal: KL1501'}
{attribute addProperty BoxType "KL1501"}
{attribute addProperty Id "StateAT %I*USINT0Data_InAT %I*ARRAY [0..1] OF UINT0CtrlAT %Q*USINT0Data_OutAT %Q*ARRAY [0..1] OF UINT0"}
{attribute addProperty CRC "1008362752"}
{attribute addProperty Size "0"}
TYPE Channel_3C1A6500 :
STRUCT
	{attribute addProperty Name "State"}
	State AT %I* : USINT;
	{attribute addProperty Name "Data_In"}
	Data_In AT %I* : ARRAY [0..1] OF UINT;
	{attribute addProperty Name "Ctrl"}
	Ctrl AT %Q* : USINT;
	{attribute addProperty Name "Data_Out"}
	Data_Out AT %Q* : ARRAY [0..1] OF UINT;
END_STRUCT
END_TYPE

// ---- DUTs/IO/PDOs/Channel_B5275D8E.TcDUT
{attribute 'GeneratedUsingTerminal: KL1501-0001'}
{attribute addProperty BoxType "KL1501-0001"}
{attribute addProperty Id "StatusAT %I*USINT0CounterAT %I*UINT0Latch_PeriodLAT %I*UINT0PeriodHAT %I*USINT0CtrlAT %Q*USINT0RegDataAT %Q*UINT0"}
{attribute addProperty CRC "3039255950"}
{attribute addProperty Size "0"}
TYPE Channel_B5275D8E :
STRUCT
	{attribute addProperty Name "Status"}
	Status AT %I* : USINT;
	{attribute addProperty Name "Counter"}
	Counter AT %I* : UINT;
	{attribute addProperty Name "Latch_PeriodL"}
	Latch_PeriodL AT %I* : UINT;
	{attribute addProperty Name "PeriodH"}
	PeriodH AT %I* : USINT;
	{attribute addProperty Name "Ctrl"}
	Ctrl AT %Q* : USINT;
	{attribute addProperty Name "RegData"}
	RegData AT %Q* : UINT;
END_STRUCT
END_TYPE

// ---- DUTs/IO/PDOs/Channel_03CEAA5E.TcDUT
{attribute 'GeneratedUsingTerminal: KL1512'}
{attribute addProperty BoxType "KL1512"}
{attribute addProperty Id "StateAT %I*USINT0Data_InAT %I*UINT0CtrlAT %Q*USINT0Data_OutAT %Q*UINT0"}
{attribute addProperty CRC "63875678"}
{attribute addProperty Size "0"}
TYPE Channel_03CEAA5E :
STRUCT
	{attribute addProperty Name "State"}
	State AT %I* : USINT;
	{attribute addProperty Name "Data_In"}
	Data_In AT %I* : UINT;
	{attribute addProperty Name "Ctrl"}
	Ctrl AT %Q* : USINT;
	{attribute addProperty Name "Data_Out"}
	Data_Out AT %Q* : UINT;
END_STRUCT
END_TYPE

// ---- DUTs/IO/PDOs/Channel_70C997F3.TcDUT
{attribute 'GeneratedUsingTerminal: KL1859'}
{attribute addProperty BoxType "KL1859"}
{attribute addProperty Id "InputAT %I*BOOL0OutputAT %Q*BOOL0"}
{attribute addProperty CRC "1892259827"}
{attribute addProperty Size "0"}
TYPE Channel_70C997F3 :
STRUCT
	{attribute addProperty Name "Input"}
	Input AT %I* : BOOL;
	{attribute addProperty Name "Output"}
	Output AT %Q* : BOOL;
END_STRUCT
END_TYPE

// ---- DUTs/IO/PDOs/Channel_1D6668A9.TcDUT
{attribute 'GeneratedUsingTerminal: KL1904'}
{attribute addProperty BoxType "KL1904"}
{attribute addProperty Id "Safety_InAT %I*ARRAY[0..5] OF BYTE0Safety_OutAT %Q*ARRAY[0..5] OF BYTE0"}
{attribute addProperty CRC "493250729"}
{attribute addProperty Size "0"}
TYPE Channel_1D6668A9 :
STRUCT
	{attribute addProperty Name "Safety_In"}
	Safety_In AT %I* : ARRAY[0..5] OF BYTE;
	{attribute addProperty Name "Safety_Out"}
	Safety_Out AT %Q* : ARRAY[0..5] OF BYTE;
END_STRUCT
END_TYPE

// ---- DUTs/IO/PDOs/Channel_6B723A16.TcDUT
{attribute 'GeneratedUsingTerminal: KL1644-0050'}
{attribute addProperty BoxType "KL1644-0050"}
{attribute addProperty Id "SwitchAT %I*BOOL0OutputAT %Q*BOOL0"}
{attribute addProperty CRC "1802648086"}
{attribute addProperty Size "0"}
TYPE Channel_6B723A16 :
STRUCT
	{attribute addProperty Name "Switch"}
	Switch AT %I* : BOOL;
	{attribute addProperty Name "Output"}
	Output AT %Q* : BOOL;
END_STRUCT
END_TYPE

// ---- DUTs/IO/PDOs/Channel_460B8C40.TcDUT
{attribute 'GeneratedUsingTerminal: KL2012'}
{attribute addProperty BoxType "KL2012"}
{attribute addProperty Id "OutputAT %Q*BOOL0"}
{attribute addProperty CRC "1175161920"}
{attribute addProperty Size "0"}
TYPE Channel_460B8C40 EXTENDS OutputBase_10CEE7DE :
STRUCT
	{attribute addProperty Name "Output"}
	Output AT %Q* : BOOL;
END_STRUCT
END_TYPE

// ---- DUTs/IO/PDOs/Channel_DCF170BB.TcDUT
{attribute 'GeneratedUsingTerminal: KL2212'}
{attribute addProperty BoxType "KL2212"}
{attribute addProperty Id "WireBreakAT %I*BOOL0CurcuitAT %I*BOOL0OutputAT %Q*BOOL0"}
{attribute addProperty CRC "3706810555"}
{attribute addProperty Size "0"}
TYPE Channel_DCF170BB :
STRUCT
	{attribute addProperty Name "WireBreak"}
	WireBreak AT %I* : BOOL;
	{attribute addProperty Name "Curcuit"}
	Curcuit AT %I* : BOOL;
	{attribute addProperty Name "Output"}
	Output AT %Q* : BOOL;
END_STRUCT
END_TYPE

// ---- DUTs/IO/PDOs/Channel_26FC8FD8.TcDUT
{attribute 'GeneratedUsingTerminal: KL2284'}
{attribute addProperty BoxType "KL2284"}
{attribute addProperty Id "CWAT %Q*BOOL0CCWAT %Q*BOOL0"}
{attribute addProperty CRC "654086104"}
{attribute addProperty Size "0"}
TYPE Channel_26FC8FD8 EXTENDS OutputBase_10CEE7DE :
STRUCT
	{attribute addProperty Name "CW"}
	CW AT %Q* : BOOL;
	{attribute addProperty Name "CCW"}
	CCW AT %Q* : BOOL;
END_STRUCT
END_TYPE

// ---- DUTs/IO/PDOs/Channel_FEA3DBF8.TcDUT
{attribute 'GeneratedUsingTerminal: KL2531'}
{attribute addProperty BoxType "KL2531"}
{attribute addProperty Id "StatusAT %I*USINT0PositionAT %I*UINT0ExtStatusAT %I*UINT0CtrlAT %Q*USINT0VelocityAT %Q*INT0ExtCtrlAT %Q*UINT0"}
{attribute addProperty CRC "4272151544"}
{attribute addProperty Size "0"}
TYPE Channel_FEA3DBF8 :
STRUCT
	{attribute addProperty Name "Status"}
	Status AT %I* : USINT;
	{attribute addProperty Name "Position"}
	Position AT %I* : UINT;
	{attribute addProperty Name "ExtStatus"}
	ExtStatus AT %I* : UINT;
	{attribute addProperty Name "Ctrl"}
	Ctrl AT %Q* : USINT;
	{attribute addProperty Name "Velocity"}
	Velocity AT %Q* : INT;
	{attribute addProperty Name "ExtCtrl"}
	ExtCtrl AT %Q* : UINT;
END_STRUCT
END_TYPE

// ---- DUTs/IO/PDOs/Channel_0D1929F0.TcDUT
{attribute 'GeneratedUsingTerminal: KL2531-0001'}
{attribute addProperty BoxType "KL2531-0001"}
{attribute addProperty Id "StatusAT %I*USINT0PositionAT %I*UDINT0ExtStatusAT %I*UINT0CtrlAT %Q*USINT0VelocityAT %Q*DINT0ExtCtrlAT %Q*UINT0"}
{attribute addProperty CRC "219752944"}
{attribute addProperty Size "0"}
TYPE Channel_0D1929F0 :
STRUCT
	{attribute addProperty Name "Status"}
	Status AT %I* : USINT;
	{attribute addProperty Name "Position"}
	Position AT %I* : UDINT;
	{attribute addProperty Name "ExtStatus"}
	ExtStatus AT %I* : UINT;
	{attribute addProperty Name "Ctrl"}
	Ctrl AT %Q* : USINT;
	{attribute addProperty Name "Velocity"}
	Velocity AT %Q* : DINT;
	{attribute addProperty Name "ExtCtrl"}
	ExtCtrl AT %Q* : UINT;
END_STRUCT
END_TYPE

// ---- DUTs/IO/PDOs/Channel_6576A681.TcDUT
{attribute 'GeneratedUsingTerminal: KL2532'}
{attribute addProperty BoxType "KL2532"}
{attribute addProperty Id "StateAT %I*USINT0Data_InAT %I*INT0CtrlAT %Q*USINT0Data_OutAT %Q*INT0"}
{attribute addProperty CRC "1702274689"}
{attribute addProperty Size "0"}
TYPE Channel_6576A681 :
STRUCT
	{attribute addProperty Name "State"}
	State AT %I* : USINT;
	{attribute addProperty Name "Data_In"}
	Data_In AT %I* : INT;
	{attribute addProperty Name "Ctrl"}
	Ctrl AT %Q* : USINT;
	{attribute addProperty Name "Data_Out"}
	Data_Out AT %Q* : INT;
END_STRUCT
END_TYPE

// ---- DUTs/IO/PDOs/Channel_2589C8DC.TcDUT
{attribute 'GeneratedUsingTerminal: KL2641'}
{attribute addProperty BoxType "KL2641"}
{attribute addProperty Id "StateAT %I*BOOL0OutputAT %Q*BOOL0"}
{attribute addProperty CRC "629786844"}
{attribute addProperty Size "0"}
TYPE Channel_2589C8DC :
STRUCT
	{attribute addProperty Name "State"}
	State AT %I* : BOOL;
	{attribute addProperty Name "Output"}
	Output AT %Q* : BOOL;
END_STRUCT
END_TYPE

// ---- DUTs/IO/PDOs/Channel_BF3661CD.TcDUT
{attribute 'GeneratedUsingTerminal: KL2641-0001'}
{attribute addProperty BoxType "KL2641-0001"}
{attribute addProperty Id "Manual_StateAT %I*BOOL0ReservedAT %I*BOOL0OutputAT %Q*BOOL0"}
{attribute addProperty CRC "3208012237"}
{attribute addProperty Size "0"}
TYPE Channel_BF3661CD :
STRUCT
	{attribute addProperty Name "Manual_State"}
	Manual_State AT %I* : BOOL;
	{attribute addProperty Name "Reserved"}
	Reserved AT %I* : BOOL;
	{attribute addProperty Name "Output"}
	Output AT %Q* : BOOL;
END_STRUCT
END_TYPE

// ---- DUTs/IO/PDOs/Channel_2EC3E8CA.TcDUT
{attribute 'GeneratedUsingTerminal: KL2819'}
{attribute addProperty BoxType "KL2819"}
{attribute addProperty Id "StatusAT %I*USINT0DiagAT %I*WORD0CtrlAT %Q*USINT0OutputAT %Q*WORD0"}
{attribute addProperty CRC "784591050"}
{attribute addProperty Size "0"}
TYPE Channel_2EC3E8CA :
STRUCT
	{attribute addProperty Name "Status"}
	Status AT %I* : USINT;
	{attribute addProperty Name "Diag"}
	Diag AT %I* : WORD;
	{attribute addProperty Name "Ctrl"}
	Ctrl AT %Q* : USINT;
	{attribute addProperty Name "Output"}
	Output AT %Q* : WORD;
END_STRUCT
END_TYPE

// ---- DUTs/IO/PDOs/Channel_F5DB8AD1.TcDUT
{attribute 'GeneratedUsingTerminal: KL2642-0050'}
{attribute addProperty BoxType "KL2642-0050"}
{attribute addProperty Id "State_RelayAT %I*BOOL0OutputAT %Q*BOOL0"}
{attribute addProperty CRC "4124805841"}
{attribute addProperty Size "0"}
TYPE Channel_F5DB8AD1 :
STRUCT
	{attribute addProperty Name "State_Relay"}
	State_Relay AT %I* : BOOL;
	{attribute addProperty Name "Output"}
	Output AT %Q* : BOOL;
END_STRUCT
END_TYPE

// ---- DUTs/IO/PDOs/Channel_6D8B740B.TcDUT
{attribute 'GeneratedUsingTerminal: KL2652-0050'}
{attribute addProperty BoxType "KL2652-0050"}
{attribute addProperty Id "State_AutoAT %I*BOOL0State_RelayAT %I*BOOL0OutputAT %Q*BOOL0"}
{attribute addProperty CRC "1837855755"}
{attribute addProperty Size "0"}
TYPE Channel_6D8B740B :
STRUCT
	{attribute addProperty Name "State_Auto"}
	State_Auto AT %I* : BOOL;
	{attribute addProperty Name "State_Relay"}
	State_Relay AT %I* : BOOL;
	{attribute addProperty Name "Output"}
	Output AT %Q* : BOOL;
END_STRUCT
END_TYPE

// ---- DUTs/IO/PDOs/Channel_2DA3FF3C.TcDUT
{attribute 'GeneratedUsingTerminal: KL3351'}
{attribute addProperty BoxType "KL3351"}
{attribute addProperty Id "StatusAT %I*USINT0Ud_RegInAT %I*INT0UrefAT %I*INT0CtrlAT %Q*USINT0RegOutAT %Q*INT0"}
{attribute addProperty CRC "765722428"}
{attribute addProperty Size "0"}
TYPE Channel_2DA3FF3C :
STRUCT
	{attribute addProperty Name "Status"}
	Status AT %I* : USINT;
	{attribute addProperty Name "Ud_RegIn"}
	Ud_RegIn AT %I* : INT;
	{attribute addProperty Name "Uref"}
	Uref AT %I* : INT;
	{attribute addProperty Name "Ctrl"}
	Ctrl AT %Q* : USINT;
	{attribute addProperty Name "RegOut"}
	RegOut AT %Q* : INT;
END_STRUCT
END_TYPE

// ---- DUTs/IO/PDOs/Channel_0514A8FA.TcDUT
{attribute 'GeneratedUsingTerminal: KL3351-0003'}
{attribute addProperty BoxType "KL3351-0003"}
{attribute addProperty Id "StatusAT %I*USINT0Ud_RegInAT %I*INT0UrefAT %I*INT0CtrlAT %Q*USINT0RegOutAT %Q*INT0Ctrl1AT %Q*USINT0"}
{attribute addProperty CRC "85240058"}
{attribute addProperty Size "0"}
TYPE Channel_0514A8FA :
STRUCT
	{attribute addProperty Name "Status"}
	Status AT %I* : USINT;
	{attribute addProperty Name "Ud_RegIn"}
	Ud_RegIn AT %I* : INT;
	{attribute addProperty Name "Uref"}
	Uref AT %I* : INT;
	{attribute addProperty Name "Ctrl"}
	Ctrl AT %Q* : USINT;
	{attribute addProperty Name "RegOut"}
	RegOut AT %Q* : INT;
	{attribute addProperty Name "Ctrl1"}
	Ctrl1 AT %Q* : USINT;
END_STRUCT
END_TYPE

// ---- DUTs/IO/PDOs/Channel_4E9D1E2D.TcDUT
{attribute 'GeneratedUsingTerminal: KL3356'}
{attribute addProperty BoxType "KL3356"}
{attribute addProperty Id "StatusAT %I*USINT0RegInAT %I*UINT0AnStatusAT %I*USINT0WeightAT %I*UINT0CtrlAT %Q*USINT0RegOutAT %Q*UINT0AnCtrlAT %Q*USINT0"}
{attribute addProperty CRC "1318919725"}
{attribute addProperty Size "0"}
TYPE Channel_4E9D1E2D :
STRUCT
	{attribute addProperty Name "Status"}
	Status AT %I* : USINT;
	{attribute addProperty Name "RegIn"}
	RegIn AT %I* : UINT;
	{attribute addProperty Name "AnStatus"}
	AnStatus AT %I* : USINT;
	{attribute addProperty Name "Weight"}
	Weight AT %I* : UINT;
	{attribute addProperty Name "Ctrl"}
	Ctrl AT %Q* : USINT;
	{attribute addProperty Name "RegOut"}
	RegOut AT %Q* : UINT;
	{attribute addProperty Name "AnCtrl"}
	AnCtrl AT %Q* : USINT;
END_STRUCT
END_TYPE

// ---- DUTs/IO/PDOs/Channel_78571FB4.TcDUT
{attribute 'GeneratedUsingTerminal: KL3361'}
{attribute addProperty BoxType "KL3361"}
{attribute addProperty Id "StateAT %I*USINT0Data_In_0AT %I*UINT0Data_In_1AT %I*UINT0Data_In_2AT %I*UINT0Data_In_3AT %I*UINT0Data_In_4AT %I*UINT0Data_In_5AT %I*UINT0Data_In_6AT %I*UINT0Data_In_7AT %I*UINT0Data_In_8AT %I*UINT0Data_In_9AT %I*UINT0Data_In_10AT %I*UINT0CtrlAT %Q*USINT0Data_Out_0AT %Q*UINT0Data_Out_1AT %Q*UINT0Data_Out_2AT %Q*UINT0Data_Out_3AT %Q*UINT0Data_Out_4AT %Q*UINT0Data_Out_5AT %Q*UINT0Data_Out_6AT %Q*UINT0Data_Out_7AT %Q*UINT0Data_Out_8AT %Q*UINT0Data_Out_9AT %Q*UINT0Data_Out_10AT %Q*UINT0"}
{attribute addProperty CRC "2018975668"}
{attribute addProperty Size "0"}
TYPE Channel_78571FB4 :
STRUCT
	{attribute addProperty Name "State"}
	State AT %I* : USINT;
	{attribute addProperty Name "Data_In_0"}
	Data_In_0 AT %I* : UINT;
	{attribute addProperty Name "Data_In_1"}
	Data_In_1 AT %I* : UINT;
	{attribute addProperty Name "Data_In_2"}
	Data_In_2 AT %I* : UINT;
	{attribute addProperty Name "Data_In_3"}
	Data_In_3 AT %I* : UINT;
	{attribute addProperty Name "Data_In_4"}
	Data_In_4 AT %I* : UINT;
	{attribute addProperty Name "Data_In_5"}
	Data_In_5 AT %I* : UINT;
	{attribute addProperty Name "Data_In_6"}
	Data_In_6 AT %I* : UINT;
	{attribute addProperty Name "Data_In_7"}
	Data_In_7 AT %I* : UINT;
	{attribute addProperty Name "Data_In_8"}
	Data_In_8 AT %I* : UINT;
	{attribute addProperty Name "Data_In_9"}
	Data_In_9 AT %I* : UINT;
	{attribute addProperty Name "Data_In_10"}
	Data_In_10 AT %I* : UINT;
	{attribute addProperty Name "Ctrl"}
	Ctrl AT %Q* : USINT;
	{attribute addProperty Name "Data_Out_0"}
	Data_Out_0 AT %Q* : UINT;
	{attribute addProperty Name "Data_Out_1"}
	Data_Out_1 AT %Q* : UINT;
	{attribute addProperty Name "Data_Out_2"}
	Data_Out_2 AT %Q* : UINT;
	{attribute addProperty Name "Data_Out_3"}
	Data_Out_3 AT %Q* : UINT;
	{attribute addProperty Name "Data_Out_4"}
	Data_Out_4 AT %Q* : UINT;
	{attribute addProperty Name "Data_Out_5"}
	Data_Out_5 AT %Q* : UINT;
	{attribute addProperty Name "Data_Out_6"}
	Data_Out_6 AT %Q* : UINT;
	{attribute addProperty Name "Data_Out_7"}
	Data_Out_7 AT %Q* : UINT;
	{attribute addProperty Name "Data_Out_8"}
	Data_Out_8 AT %Q* : UINT;
	{attribute addProperty Name "Data_Out_9"}
	Data_Out_9 AT %Q* : UINT;
	{attribute addProperty Name "Data_Out_10"}
	Data_Out_10 AT %Q* : UINT;
END_STRUCT
END_TYPE

// ---- DUTs/IO/PDOs/Channel_87905831.TcDUT
{attribute 'GeneratedUsingTerminal: KL6211'}
{attribute addProperty BoxType "KL6211"}
{attribute addProperty Id "StatusAT %I*UINT0Parameter_InAT %I*UDINT0ASI_In_Slave_1_StatusAT %I*USINT0ASI_In_Slave_3_Slave_2AT %I*USINT0ASI_In_Slave_5_Slave_4AT %I*USINT0ASI_In_Slave_7_Slave_6AT %I*USINT0ASI_In_Slave_9_Slave_8AT %I*USINT0ASI_In_Slave_11_Slave_10AT %I*USINT0ControlAT %Q*UINT0Parameter_OutAT %Q*UDINT0ASI_Out_Slave_1_ControlAT %Q*USINT0ASI_Out_Slave_3_Slave_2AT %Q*USINT0ASI_Out_Slave_5_Slave_4AT %Q*USINT0ASI_Out_Slave_7_Slave_6AT %Q*USINT0ASI_Out_Slave_9_Slave_8AT %Q*USINT0ASI_Out_Slave_11_Slave_10AT %Q*USINT0"}
{attribute addProperty CRC "2274383921"}
{attribute addProperty Size "0"}
TYPE Channel_87905831 :
STRUCT
	{attribute addProperty Name "Status"}
	Status AT %I* : UINT;
	{attribute addProperty Name "Parameter_In"}
	Parameter_In AT %I* : UDINT;
	{attribute addProperty Name "ASI_In_Slave_1_Status"}
	ASI_In_Slave_1_Status AT %I* : USINT;
	{attribute addProperty Name "ASI_In_Slave_3_Slave_2"}
	ASI_In_Slave_3_Slave_2 AT %I* : USINT;
	{attribute addProperty Name "ASI_In_Slave_5_Slave_4"}
	ASI_In_Slave_5_Slave_4 AT %I* : USINT;
	{attribute addProperty Name "ASI_In_Slave_7_Slave_6"}
	ASI_In_Slave_7_Slave_6 AT %I* : USINT;
	{attribute addProperty Name "ASI_In_Slave_9_Slave_8"}
	ASI_In_Slave_9_Slave_8 AT %I* : USINT;
	{attribute addProperty Name "ASI_In_Slave_11_Slave_10"}
	ASI_In_Slave_11_Slave_10 AT %I* : USINT;
	{attribute addProperty Name "Control"}
	Control AT %Q* : UINT;
	{attribute addProperty Name "Parameter_Out"}
	Parameter_Out AT %Q* : UDINT;
	{attribute addProperty Name "ASI_Out_Slave_1_Control"}
	ASI_Out_Slave_1_Control AT %Q* : USINT;
	{attribute addProperty Name "ASI_Out_Slave_3_Slave_2"}
	ASI_Out_Slave_3_Slave_2 AT %Q* : USINT;
	{attribute addProperty Name "ASI_Out_Slave_5_Slave_4"}
	ASI_Out_Slave_5_Slave_4 AT %Q* : USINT;
	{attribute addProperty Name "ASI_Out_Slave_7_Slave_6"}
	ASI_Out_Slave_7_Slave_6 AT %Q* : USINT;
	{attribute addProperty Name "ASI_Out_Slave_9_Slave_8"}
	ASI_Out_Slave_9_Slave_8 AT %Q* : USINT;
	{attribute addProperty Name "ASI_Out_Slave_11_Slave_10"}
	ASI_Out_Slave_11_Slave_10 AT %Q* : USINT;
END_STRUCT
END_TYPE

// ---- DUTs/IO/PDOs/Channel_099BCCDA.TcDUT
{attribute 'GeneratedUsingTerminal: KL6211-0020'}
{attribute addProperty BoxType "KL6211-0020"}
{attribute addProperty Id "StatusAT %I*UINT0Parameter_InAT %I*UDINT0ASI_In_StatusAT %I*BYTE0ASI_In_Slave_1AT %I*BYTE0ASI_In_Slave_2AT %I*BYTE0ASI_In_Slave_3AT %I*BYTE0ASI_In_Slave_4AT %I*BYTE0ASI_In_Slave_5AT %I*BYTE0ASI_In_Slave_6AT %I*BYTE0ASI_In_Slave_7AT %I*BYTE0ASI_In_Slave_8AT %I*BYTE0ASI_In_Slave_9AT %I*BYTE0ASI_In_Slave_10AT %I*BYTE0ASI_In_Slave_11AT %I*BYTE0ControlAT %Q*UINT0Parameter_OutAT %Q*UDINT0ASI_Out_ControlAT %Q*BYTE0ASI_Out_Slave_1AT %Q*BYTE0ASI_Out_Slave_2AT %Q*BYTE0ASI_Out_Slave_3AT %Q*BYTE0ASI_Out_Slave_4AT %Q*BYTE0ASI_Out_Slave_5AT %Q*BYTE0ASI_Out_Slave_6AT %Q*BYTE0ASI_Out_Slave_7AT %Q*BYTE0ASI_Out_Slave_8AT %Q*BYTE0ASI_Out_Slave_9AT %Q*BYTE0ASI_Out_Slave_10AT %Q*BYTE0ASI_Out_Slave_11AT %Q*BYTE0"}
{attribute addProperty CRC "161205466"}
{attribute addProperty Size "0"}
TYPE Channel_099BCCDA :
STRUCT
	{attribute addProperty Name "Status"}
	Status AT %I* : UINT;
	{attribute addProperty Name "Parameter_In"}
	Parameter_In AT %I* : UDINT;
	{attribute addProperty Name "ASI_In_Status"}
	ASI_In_Status AT %I* : BYTE;
	{attribute addProperty Name "ASI_In_Slave_1"}
	ASI_In_Slave_1 AT %I* : BYTE;
	{attribute addProperty Name "ASI_In_Slave_2"}
	ASI_In_Slave_2 AT %I* : BYTE;
	{attribute addProperty Name "ASI_In_Slave_3"}
	ASI_In_Slave_3 AT %I* : BYTE;
	{attribute addProperty Name "ASI_In_Slave_4"}
	ASI_In_Slave_4 AT %I* : BYTE;
	{attribute addProperty Name "ASI_In_Slave_5"}
	ASI_In_Slave_5 AT %I* : BYTE;
	{attribute addProperty Name "ASI_In_Slave_6"}
	ASI_In_Slave_6 AT %I* : BYTE;
	{attribute addProperty Name "ASI_In_Slave_7"}
	ASI_In_Slave_7 AT %I* : BYTE;
	{attribute addProperty Name "ASI_In_Slave_8"}
	ASI_In_Slave_8 AT %I* : BYTE;
	{attribute addProperty Name "ASI_In_Slave_9"}
	ASI_In_Slave_9 AT %I* : BYTE;
	{attribute addProperty Name "ASI_In_Slave_10"}
	ASI_In_Slave_10 AT %I* : BYTE;
	{attribute addProperty Name "ASI_In_Slave_11"}
	ASI_In_Slave_11 AT %I* : BYTE;
	{attribute addProperty Name "Control"}
	Control AT %Q* : UINT;
	{attribute addProperty Name "Parameter_Out"}
	Parameter_Out AT %Q* : UDINT;
	{attribute addProperty Name "ASI_Out_Control"}
	ASI_Out_Control AT %Q* : BYTE;
	{attribute addProperty Name "ASI_Out_Slave_1"}
	ASI_Out_Slave_1 AT %Q* : BYTE;
	{attribute addProperty Name "ASI_Out_Slave_2"}
	ASI_Out_Slave_2 AT %Q* : BYTE;
	{attribute addProperty Name "ASI_Out_Slave_3"}
	ASI_Out_Slave_3 AT %Q* : BYTE;
	{attribute addProperty Name "ASI_Out_Slave_4"}
	ASI_Out_Slave_4 AT %Q* : BYTE;
	{attribute addProperty Name "ASI_Out_Slave_5"}
	ASI_Out_Slave_5 AT %Q* : BYTE;
	{attribute addProperty Name "ASI_Out_Slave_6"}
	ASI_Out_Slave_6 AT %Q* : BYTE;
	{attribute addProperty Name "ASI_Out_Slave_7"}
	ASI_Out_Slave_7 AT %Q* : BYTE;
	{attribute addProperty Name "ASI_Out_Slave_8"}
	ASI_Out_Slave_8 AT %Q* : BYTE;
	{attribute addProperty Name "ASI_Out_Slave_9"}
	ASI_Out_Slave_9 AT %Q* : BYTE;
	{attribute addProperty Name "ASI_Out_Slave_10"}
	ASI_Out_Slave_10 AT %Q* : BYTE;
	{attribute addProperty Name "ASI_Out_Slave_11"}
	ASI_Out_Slave_11 AT %Q* : BYTE;
END_STRUCT
END_TYPE

// ---- DUTs/IO/PDOs/Channel_82ADD076.TcDUT
{attribute 'GeneratedUsingTerminal: KL6211-0002'}
{attribute addProperty BoxType "KL6211-0002"}
{attribute addProperty Id "StatusAT %I*UINT0Parameter_InAT %I*UDINT0ASI_In_Slave_1_StatusAT %I*USINT0ASI_In_Slave_3_Slave_2AT %I*USINT0ASI_In_Slave_5_Slave_4AT %I*USINT0ASI_In_Slave_7_Slave_6AT %I*USINT0ASI_In_Slave_9_Slave_8AT %I*USINT0ASI_In_Slave_11_Slave_10AT %I*USINT0ASI_In_Slave_13_Slave_12AT %I*USINT0ASI_In_Slave_15_Slave_14AT %I*USINT0ASI_In_Slave_17_Slave_16AT %I*USINT0ASI_In_Slave_19_Slave_18AT %I*USINT0ASI_In_Slave_21_Slave_20AT %I*USINT0ASI_In_Slave_23_Slave_22AT %I*USINT0ASI_In_Slave_25_Slave_24AT %I*USINT0ASI_In_Slave_27_Slave_26AT %I*USINT0ASI_In_Slave_29_Slave_28AT %I*USINT0ASI_In_Slave_31_Slave_30AT %I*USINT0ControlAT %Q*UINT0Parameter_OutAT %Q*UDINT0ASI_Out_Slave_1_ControlAT %Q*USINT0ASI_Out_Slave_3_Slave_2AT %Q*USINT0ASI_Out_Slave_5_Slave_4AT %Q*USINT0ASI_Out_Slave_7_Slave_6AT %Q*USINT0ASI_Out_Slave_9_Slave_8AT %Q*USINT0ASI_Out_Slave_11_Slave_10AT %Q*USINT0ASI_Out_Slave_13_Slave_12AT %Q*USINT0ASI_Out_Slave_15_Slave_14AT %Q*USINT0ASI_Out_Slave_17_Slave_16AT %Q*USINT0ASI_Out_Slave_19_Slave_18AT %Q*USINT0ASI_Out_Slave_21_Slave_20AT %Q*USINT0ASI_Out_Slave_23_Slave_22AT %Q*USINT0ASI_Out_Slave_25_Slave_24AT %Q*USINT0ASI_Out_Slave_27_Slave_26AT %Q*USINT0ASI_Out_Slave_29_Slave_28AT %Q*USINT0ASI_Out_Slave_31_Slave_30AT %Q*USINT0"}
{attribute addProperty CRC "2192429174"}
{attribute addProperty Size "0"}
TYPE Channel_82ADD076 :
STRUCT
	{attribute addProperty Name "Status"}
	Status AT %I* : UINT;
	{attribute addProperty Name "Parameter_In"}
	Parameter_In AT %I* : UDINT;
	{attribute addProperty Name "ASI_In_Slave_1_Status"}
	ASI_In_Slave_1_Status AT %I* : USINT;
	{attribute addProperty Name "ASI_In_Slave_3_Slave_2"}
	ASI_In_Slave_3_Slave_2 AT %I* : USINT;
	{attribute addProperty Name "ASI_In_Slave_5_Slave_4"}
	ASI_In_Slave_5_Slave_4 AT %I* : USINT;
	{attribute addProperty Name "ASI_In_Slave_7_Slave_6"}
	ASI_In_Slave_7_Slave_6 AT %I* : USINT;
	{attribute addProperty Name "ASI_In_Slave_9_Slave_8"}
	ASI_In_Slave_9_Slave_8 AT %I* : USINT;
	{attribute addProperty Name "ASI_In_Slave_11_Slave_10"}
	ASI_In_Slave_11_Slave_10 AT %I* : USINT;
	{attribute addProperty Name "ASI_In_Slave_13_Slave_12"}
	ASI_In_Slave_13_Slave_12 AT %I* : USINT;
	{attribute addProperty Name "ASI_In_Slave_15_Slave_14"}
	ASI_In_Slave_15_Slave_14 AT %I* : USINT;
	{attribute addProperty Name "ASI_In_Slave_17_Slave_16"}
	ASI_In_Slave_17_Slave_16 AT %I* : USINT;
	{attribute addProperty Name "ASI_In_Slave_19_Slave_18"}
	ASI_In_Slave_19_Slave_18 AT %I* : USINT;
	{attribute addProperty Name "ASI_In_Slave_21_Slave_20"}
	ASI_In_Slave_21_Slave_20 AT %I* : USINT;
	{attribute addProperty Name "ASI_In_Slave_23_Slave_22"}
	ASI_In_Slave_23_Slave_22 AT %I* : USINT;
	{attribute addProperty Name "ASI_In_Slave_25_Slave_24"}
	ASI_In_Slave_25_Slave_24 AT %I* : USINT;
	{attribute addProperty Name "ASI_In_Slave_27_Slave_26"}
	ASI_In_Slave_27_Slave_26 AT %I* : USINT;
	{attribute addProperty Name "ASI_In_Slave_29_Slave_28"}
	ASI_In_Slave_29_Slave_28 AT %I* : USINT;
	{attribute addProperty Name "ASI_In_Slave_31_Slave_30"}
	ASI_In_Slave_31_Slave_30 AT %I* : USINT;
	{attribute addProperty Name "Control"}
	Control AT %Q* : UINT;
	{attribute addProperty Name "Parameter_Out"}
	Parameter_Out AT %Q* : UDINT;
	{attribute addProperty Name "ASI_Out_Slave_1_Control"}
	ASI_Out_Slave_1_Control AT %Q* : USINT;
	{attribute addProperty Name "ASI_Out_Slave_3_Slave_2"}
	ASI_Out_Slave_3_Slave_2 AT %Q* : USINT;
	{attribute addProperty Name "ASI_Out_Slave_5_Slave_4"}
	ASI_Out_Slave_5_Slave_4 AT %Q* : USINT;
	{attribute addProperty Name "ASI_Out_Slave_7_Slave_6"}
	ASI_Out_Slave_7_Slave_6 AT %Q* : USINT;
	{attribute addProperty Name "ASI_Out_Slave_9_Slave_8"}
	ASI_Out_Slave_9_Slave_8 AT %Q* : USINT;
	{attribute addProperty Name "ASI_Out_Slave_11_Slave_10"}
	ASI_Out_Slave_11_Slave_10 AT %Q* : USINT;
	{attribute addProperty Name "ASI_Out_Slave_13_Slave_12"}
	ASI_Out_Slave_13_Slave_12 AT %Q* : USINT;
	{attribute addProperty Name "ASI_Out_Slave_15_Slave_14"}
	ASI_Out_Slave_15_Slave_14 AT %Q* : USINT;
	{attribute addProperty Name "ASI_Out_Slave_17_Slave_16"}
	ASI_Out_Slave_17_Slave_16 AT %Q* : USINT;
	{attribute addProperty Name "ASI_Out_Slave_19_Slave_18"}
	ASI_Out_Slave_19_Slave_18 AT %Q* : USINT;
	{attribute addProperty Name "ASI_Out_Slave_21_Slave_20"}
	ASI_Out_Slave_21_Slave_20 AT %Q* : USINT;
	{attribute addProperty Name "ASI_Out_Slave_23_Slave_22"}
	ASI_Out_Slave_23_Slave_22 AT %Q* : USINT;
	{attribute addProperty Name "ASI_Out_Slave_25_Slave_24"}
	ASI_Out_Slave_25_Slave_24 AT %Q* : USINT;
	{attribute addProperty Name "ASI_Out_Slave_27_Slave_26"}
	ASI_Out_Slave_27_Slave_26 AT %Q* : USINT;
	{attribute addProperty Name "ASI_Out_Slave_29_Slave_28"}
	ASI_Out_Slave_29_Slave_28 AT %Q* : USINT;
	{attribute addProperty Name "ASI_Out_Slave_31_Slave_30"}
	ASI_Out_Slave_31_Slave_30 AT %Q* : USINT;
END_STRUCT
END_TYPE

// ---- DUTs/IO/PDOs/Channel_332F026B.TcDUT
{attribute 'GeneratedUsingTerminal: KL6211-0022'}
{attribute addProperty BoxType "KL6211-0022"}
{attribute addProperty Id "StatusAT %I*UINT0Parameter_InAT %I*UDINT0ASI_In_StatusAT %I*BYTE0ASI_In_Slave_1AT %I*BYTE0ASI_In_Slave_2AT %I*BYTE0ASI_In_Slave_3AT %I*BYTE0ASI_In_Slave_4AT %I*BYTE0ASI_In_Slave_5AT %I*BYTE0ASI_In_Slave_6AT %I*BYTE0ASI_In_Slave_7AT %I*BYTE0ASI_In_Slave_8AT %I*BYTE0ASI_In_Slave_9AT %I*BYTE0ASI_In_Slave_10AT %I*BYTE0ASI_In_Slave_11AT %I*BYTE0ASI_In_Slave_12AT %I*BYTE0ASI_In_Slave_13AT %I*BYTE0ASI_In_Slave_14AT %I*BYTE0ASI_In_Slave_15AT %I*BYTE0ASI_In_Slave_16AT %I*BYTE0ASI_In_Slave_17AT %I*BYTE0ASI_In_Slave_18AT %I*BYTE0ASI_In_Slave_19AT %I*BYTE0ASI_In_Slave_20AT %I*BYTE0ASI_In_Slave_21AT %I*BYTE0ASI_In_Slave_22AT %I*BYTE0ASI_In_Slave_23AT %I*BYTE0ASI_In_Slave_24AT %I*BYTE0ASI_In_Slave_25AT %I*BYTE0ASI_In_Slave_26AT %I*BYTE0ASI_In_Slave_27AT %I*BYTE0ASI_In_Slave_28AT %I*BYTE0ASI_In_Slave_29AT %I*BYTE0ASI_In_Slave_30AT %I*BYTE0ASI_In_Slave_31AT %I*BYTE0ControlAT %Q*UINT0Parameter_OutAT %Q*UDINT0ASI_Out_ControlAT %Q*BYTE0ASI_Out_Slave_1AT %Q*BYTE0ASI_Out_Slave_2AT %Q*BYTE0ASI_Out_Slave_3AT %Q*BYTE0ASI_Out_Slave_4AT %Q*BYTE0ASI_Out_Slave_5AT %Q*BYTE0ASI_Out_Slave_6AT %Q*BYTE0ASI_Out_Slave_7AT %Q*BYTE0ASI_Out_Slave_8AT %Q*BYTE0ASI_Out_Slave_9AT %Q*BYTE0ASI_Out_Slave_10AT %Q*BYTE0ASI_Out_Slave_11AT %Q*BYTE0ASI_Out_Slave_12AT %Q*BYTE0ASI_Out_Slave_13AT %Q*BYTE0ASI_Out_Slave_14AT %Q*BYTE0ASI_Out_Slave_15AT %Q*BYTE0ASI_Out_Slave_16AT %Q*BYTE0ASI_Out_Slave_17AT %Q*BYTE0ASI_Out_Slave_18AT %Q*BYTE0ASI_Out_Slave_19AT %Q*BYTE0ASI_Out_Slave_20AT %Q*BYTE0ASI_Out_Slave_21AT %Q*BYTE0ASI_Out_Slave_22AT %Q*BYTE0ASI_Out_Slave_23AT %Q*BYTE0ASI_Out_Slave_24AT %Q*BYTE0ASI_Out_Slave_25AT %Q*BYTE0ASI_Out_Slave_26AT %Q*BYTE0ASI_Out_Slave_27AT %Q*BYTE0ASI_Out_Slave_28AT %Q*BYTE0ASI_Out_Slave_29AT %Q*BYTE0ASI_Out_Slave_30AT %Q*BYTE0ASI_Out_Slave_31AT %Q*BYTE0"}
{attribute addProperty CRC "858718827"}
{attribute addProperty Size "0"}
TYPE Channel_332F026B :
STRUCT
	{attribute addProperty Name "Status"}
	Status AT %I* : UINT;
	{attribute addProperty Name "Parameter_In"}
	Parameter_In AT %I* : UDINT;
	{attribute addProperty Name "ASI_In_Status"}
	ASI_In_Status AT %I* : BYTE;
	{attribute addProperty Name "ASI_In_Slave_1"}
	ASI_In_Slave_1 AT %I* : BYTE;
	{attribute addProperty Name "ASI_In_Slave_2"}
	ASI_In_Slave_2 AT %I* : BYTE;
	{attribute addProperty Name "ASI_In_Slave_3"}
	ASI_In_Slave_3 AT %I* : BYTE;
	{attribute addProperty Name "ASI_In_Slave_4"}
	ASI_In_Slave_4 AT %I* : BYTE;
	{attribute addProperty Name "ASI_In_Slave_5"}
	ASI_In_Slave_5 AT %I* : BYTE;
	{attribute addProperty Name "ASI_In_Slave_6"}
	ASI_In_Slave_6 AT %I* : BYTE;
	{attribute addProperty Name "ASI_In_Slave_7"}
	ASI_In_Slave_7 AT %I* : BYTE;
	{attribute addProperty Name "ASI_In_Slave_8"}
	ASI_In_Slave_8 AT %I* : BYTE;
	{attribute addProperty Name "ASI_In_Slave_9"}
	ASI_In_Slave_9 AT %I* : BYTE;
	{attribute addProperty Name "ASI_In_Slave_10"}
	ASI_In_Slave_10 AT %I* : BYTE;
	{attribute addProperty Name "ASI_In_Slave_11"}
	ASI_In_Slave_11 AT %I* : BYTE;
	{attribute addProperty Name "ASI_In_Slave_12"}
	ASI_In_Slave_12 AT %I* : BYTE;
	{attribute addProperty Name "ASI_In_Slave_13"}
	ASI_In_Slave_13 AT %I* : BYTE;
	{attribute addProperty Name "ASI_In_Slave_14"}
	ASI_In_Slave_14 AT %I* : BYTE;
	{attribute addProperty Name "ASI_In_Slave_15"}
	ASI_In_Slave_15 AT %I* : BYTE;
	{attribute addProperty Name "ASI_In_Slave_16"}
	ASI_In_Slave_16 AT %I* : BYTE;
	{attribute addProperty Name "ASI_In_Slave_17"}
	ASI_In_Slave_17 AT %I* : BYTE;
	{attribute addProperty Name "ASI_In_Slave_18"}
	ASI_In_Slave_18 AT %I* : BYTE;
	{attribute addProperty Name "ASI_In_Slave_19"}
	ASI_In_Slave_19 AT %I* : BYTE;
	{attribute addProperty Name "ASI_In_Slave_20"}
	ASI_In_Slave_20 AT %I* : BYTE;
	{attribute addProperty Name "ASI_In_Slave_21"}
	ASI_In_Slave_21 AT %I* : BYTE;
	{attribute addProperty Name "ASI_In_Slave_22"}
	ASI_In_Slave_22 AT %I* : BYTE;
	{attribute addProperty Name "ASI_In_Slave_23"}
	ASI_In_Slave_23 AT %I* : BYTE;
	{attribute addProperty Name "ASI_In_Slave_24"}
	ASI_In_Slave_24 AT %I* : BYTE;
	{attribute addProperty Name "ASI_In_Slave_25"}
	ASI_In_Slave_25 AT %I* : BYTE;
	{attribute addProperty Name "ASI_In_Slave_26"}
	ASI_In_Slave_26 AT %I* : BYTE;
	{attribute addProperty Name "ASI_In_Slave_27"}
	ASI_In_Slave_27 AT %I* : BYTE;
	{attribute addProperty Name "ASI_In_Slave_28"}
	ASI_In_Slave_28 AT %I* : BYTE;
	{attribute addProperty Name "ASI_In_Slave_29"}
	ASI_In_Slave_29 AT %I* : BYTE;
	{attribute addProperty Name "ASI_In_Slave_30"}
	ASI_In_Slave_30 AT %I* : BYTE;
	{attribute addProperty Name "ASI_In_Slave_31"}
	ASI_In_Slave_31 AT %I* : BYTE;
	{attribute addProperty Name "Control"}
	Control AT %Q* : UINT;
	{attribute addProperty Name "Parameter_Out"}
	Parameter_Out AT %Q* : UDINT;
	{attribute addProperty Name "ASI_Out_Control"}
	ASI_Out_Control AT %Q* : BYTE;
	{attribute addProperty Name "ASI_Out_Slave_1"}
	ASI_Out_Slave_1 AT %Q* : BYTE;
	{attribute addProperty Name "ASI_Out_Slave_2"}
	ASI_Out_Slave_2 AT %Q* : BYTE;
	{attribute addProperty Name "ASI_Out_Slave_3"}
	ASI_Out_Slave_3 AT %Q* : BYTE;
	{attribute addProperty Name "ASI_Out_Slave_4"}
	ASI_Out_Slave_4 AT %Q* : BYTE;
	{attribute addProperty Name "ASI_Out_Slave_5"}
	ASI_Out_Slave_5 AT %Q* : BYTE;
	{attribute addProperty Name "ASI_Out_Slave_6"}
	ASI_Out_Slave_6 AT %Q* : BYTE;
	{attribute addProperty Name "ASI_Out_Slave_7"}
	ASI_Out_Slave_7 AT %Q* : BYTE;
	{attribute addProperty Name "ASI_Out_Slave_8"}
	ASI_Out_Slave_8 AT %Q* : BYTE;
	{attribute addProperty Name "ASI_Out_Slave_9"}
	ASI_Out_Slave_9 AT %Q* : BYTE;
	{attribute addProperty Name "ASI_Out_Slave_10"}
	ASI_Out_Slave_10 AT %Q* : BYTE;
	{attribute addProperty Name "ASI_Out_Slave_11"}
	ASI_Out_Slave_11 AT %Q* : BYTE;
	{attribute addProperty Name "ASI_Out_Slave_12"}
	ASI_Out_Slave_12 AT %Q* : BYTE;
	{attribute addProperty Name "ASI_Out_Slave_13"}
	ASI_Out_Slave_13 AT %Q* : BYTE;
	{attribute addProperty Name "ASI_Out_Slave_14"}
	ASI_Out_Slave_14 AT %Q* : BYTE;
	{attribute addProperty Name "ASI_Out_Slave_15"}
	ASI_Out_Slave_15 AT %Q* : BYTE;
	{attribute addProperty Name "ASI_Out_Slave_16"}
	ASI_Out_Slave_16 AT %Q* : BYTE;
	{attribute addProperty Name "ASI_Out_Slave_17"}
	ASI_Out_Slave_17 AT %Q* : BYTE;
	{attribute addProperty Name "ASI_Out_Slave_18"}
	ASI_Out_Slave_18 AT %Q* : BYTE;
	{attribute addProperty Name "ASI_Out_Slave_19"}
	ASI_Out_Slave_19 AT %Q* : BYTE;
	{attribute addProperty Name "ASI_Out_Slave_20"}
	ASI_Out_Slave_20 AT %Q* : BYTE;
	{attribute addProperty Name "ASI_Out_Slave_21"}
	ASI_Out_Slave_21 AT %Q* : BYTE;
	{attribute addProperty Name "ASI_Out_Slave_22"}
	ASI_Out_Slave_22 AT %Q* : BYTE;
	{attribute addProperty Name "ASI_Out_Slave_23"}
	ASI_Out_Slave_23 AT %Q* : BYTE;
	{attribute addProperty Name "ASI_Out_Slave_24"}
	ASI_Out_Slave_24 AT %Q* : BYTE;
	{attribute addProperty Name "ASI_Out_Slave_25"}
	ASI_Out_Slave_25 AT %Q* : BYTE;
	{attribute addProperty Name "ASI_Out_Slave_26"}
	ASI_Out_Slave_26 AT %Q* : BYTE;
	{attribute addProperty Name "ASI_Out_Slave_27"}
	ASI_Out_Slave_27 AT %Q* : BYTE;
	{attribute addProperty Name "ASI_Out_Slave_28"}
	ASI_Out_Slave_28 AT %Q* : BYTE;
	{attribute addProperty Name "ASI_Out_Slave_29"}
	ASI_Out_Slave_29 AT %Q* : BYTE;
	{attribute addProperty Name "ASI_Out_Slave_30"}
	ASI_Out_Slave_30 AT %Q* : BYTE;
	{attribute addProperty Name "ASI_Out_Slave_31"}
	ASI_Out_Slave_31 AT %Q* : BYTE;
END_STRUCT
END_TYPE

// ---- DUTs/IO/PDOs/Channel_A6A8AB45.TcDUT
{attribute 'GeneratedUsingTerminal: KL6211-0004'}
{attribute addProperty BoxType "KL6211-0004"}
{attribute addProperty Id "StatusAT %I*UINT0Parameter_InAT %I*UDINT0ASI_In_Slave_1_StatusAT %I*USINT0ASI_In_Slave_3_Slave_2AT %I*USINT0ASI_In_Slave_5_Slave_4AT %I*USINT0ASI_In_Slave_7_Slave_6AT %I*USINT0ASI_In_Slave_9_Slave_8AT %I*USINT0ASI_In_Slave_11_Slave_10AT %I*USINT0ASI_In_Slave_13_Slave_12AT %I*USINT0ASI_In_Slave_15_Slave_14AT %I*USINT0ASI_In_Slave_17_Slave_16AT %I*USINT0ASI_In_Slave_19_Slave_18AT %I*USINT0ASI_In_Slave_21_Slave_20AT %I*USINT0ASI_In_Slave_23_Slave_22AT %I*USINT0ASI_In_Slave_25_Slave_24AT %I*USINT0ASI_In_Slave_27_Slave_26AT %I*USINT0ASI_In_Slave_29_Slave_28AT %I*USINT0ASI_In_Slave_31_Slave_30AT %I*USINT0ASI_In_Slave_33_Slave_32AT %I*USINT0ASI_In_Slave_35_Slave_34AT %I*USINT0ASI_In_Slave_37_Slave_36AT %I*USINT0ASI_In_Slave_39_Slave_38AT %I*USINT0ASI_In_Slave_41_Slave_40AT %I*USINT0ASI_In_Slave_43_Slave_42AT %I*USINT0ASI_In_Slave_45_Slave_44AT %I*USINT0ASI_In_Slave_47_Slave_46AT %I*USINT0ASI_In_Slave_49_Slave_48AT %I*USINT0ASI_In_Slave_51_Slave_50AT %I*USINT0ASI_In_Slave_53_Slave_52AT %I*USINT0ASI_In_Slave_55_Slave_54AT %I*USINT0ASI_In_Slave_57_Slave_56AT %I*USINT0ASI_In_Slave_59_Slave_58AT %I*USINT0ASI_In_Slave_61_Slave_60AT %I*USINT0ASI_In_Slave_63_Slave_62AT %I*USINT0ControlAT %Q*UINT0Parameter_OutAT %Q*UDINT0ASI_Out_Slave_1_ControlAT %Q*USINT0ASI_Out_Slave_3_Slave_2AT %Q*USINT0ASI_Out_Slave_5_Slave_4AT %Q*USINT0ASI_Out_Slave_7_Slave_6AT %Q*USINT0ASI_Out_Slave_9_Slave_8AT %Q*USINT0ASI_Out_Slave_11_Slave_10AT %Q*USINT0ASI_Out_Slave_13_Slave_12AT %Q*USINT0ASI_Out_Slave_15_Slave_14AT %Q*USINT0ASI_Out_Slave_17_Slave_16AT %Q*USINT0ASI_Out_Slave_19_Slave_18AT %Q*USINT0ASI_Out_Slave_21_Slave_20AT %Q*USINT0ASI_Out_Slave_23_Slave_22AT %Q*USINT0ASI_Out_Slave_25_Slave_24AT %Q*USINT0ASI_Out_Slave_27_Slave_26AT %Q*USINT0ASI_Out_Slave_29_Slave_28AT %Q*USINT0ASI_Out_Slave_31_Slave_30AT %Q*USINT0ASI_Out_Slave_33_Slave_32AT %Q*USINT0ASI_Out_Slave_35_Slave_34AT %Q*USINT0ASI_Out_Slave_37_Slave_36AT %Q*USINT0ASI_Out_Slave_39_Slave_38AT %Q*USINT0ASI_Out_Slave_41_Slave_40AT %Q*USINT0ASI_Out_Slave_43_Slave_42AT %Q*USINT0ASI_Out_Slave_45_Slave_44AT %Q*USINT0ASI_Out_Slave_47_Slave_46AT %Q*USINT0ASI_Out_Slave_49_Slave_48AT %Q*USINT0ASI_Out_Slave_51_Slave_50AT %Q*USINT0ASI_Out_Slave_53_Slave_52AT %Q*USINT0ASI_Out_Slave_55_Slave_54AT %Q*USINT0ASI_Out_Slave_57_Slave_56AT %Q*USINT0ASI_Out_Slave_59_Slave_58AT %Q*USINT0ASI_Out_Slave_61_Slave_60AT %Q*USINT0ASI_Out_Slave_63_Slave_62AT %Q*USINT0"}
{attribute addProperty CRC "2796071749"}
{attribute addProperty Size "0"}
TYPE Channel_A6A8AB45 :
STRUCT
	{attribute addProperty Name "Status"}
	Status AT %I* : UINT;
	{attribute addProperty Name "Parameter_In"}
	Parameter_In AT %I* : UDINT;
	{attribute addProperty Name "ASI_In_Slave_1_Status"}
	ASI_In_Slave_1_Status AT %I* : USINT;
	{attribute addProperty Name "ASI_In_Slave_3_Slave_2"}
	ASI_In_Slave_3_Slave_2 AT %I* : USINT;
	{attribute addProperty Name "ASI_In_Slave_5_Slave_4"}
	ASI_In_Slave_5_Slave_4 AT %I* : USINT;
	{attribute addProperty Name "ASI_In_Slave_7_Slave_6"}
	ASI_In_Slave_7_Slave_6 AT %I* : USINT;
	{attribute addProperty Name "ASI_In_Slave_9_Slave_8"}
	ASI_In_Slave_9_Slave_8 AT %I* : USINT;
	{attribute addProperty Name "ASI_In_Slave_11_Slave_10"}
	ASI_In_Slave_11_Slave_10 AT %I* : USINT;
	{attribute addProperty Name "ASI_In_Slave_13_Slave_12"}
	ASI_In_Slave_13_Slave_12 AT %I* : USINT;
	{attribute addProperty Name "ASI_In_Slave_15_Slave_14"}
	ASI_In_Slave_15_Slave_14 AT %I* : USINT;
	{attribute addProperty Name "ASI_In_Slave_17_Slave_16"}
	ASI_In_Slave_17_Slave_16 AT %I* : USINT;
	{attribute addProperty Name "ASI_In_Slave_19_Slave_18"}
	ASI_In_Slave_19_Slave_18 AT %I* : USINT;
	{attribute addProperty Name "ASI_In_Slave_21_Slave_20"}
	ASI_In_Slave_21_Slave_20 AT %I* : USINT;
	{attribute addProperty Name "ASI_In_Slave_23_Slave_22"}
	ASI_In_Slave_23_Slave_22 AT %I* : USINT;
	{attribute addProperty Name "ASI_In_Slave_25_Slave_24"}
	ASI_In_Slave_25_Slave_24 AT %I* : USINT;
	{attribute addProperty Name "ASI_In_Slave_27_Slave_26"}
	ASI_In_Slave_27_Slave_26 AT %I* : USINT;
	{attribute addProperty Name "ASI_In_Slave_29_Slave_28"}
	ASI_In_Slave_29_Slave_28 AT %I* : USINT;
	{attribute addProperty Name "ASI_In_Slave_31_Slave_30"}
	ASI_In_Slave_31_Slave_30 AT %I* : USINT;
	{attribute addProperty Name "ASI_In_Slave_33_Slave_32"}
	ASI_In_Slave_33_Slave_32 AT %I* : USINT;
	{attribute addProperty Name "ASI_In_Slave_35_Slave_34"}
	ASI_In_Slave_35_Slave_34 AT %I* : USINT;
	{attribute addProperty Name "ASI_In_Slave_37_Slave_36"}
	ASI_In_Slave_37_Slave_36 AT %I* : USINT;
	{attribute addProperty Name "ASI_In_Slave_39_Slave_38"}
	ASI_In_Slave_39_Slave_38 AT %I* : USINT;
	{attribute addProperty Name "ASI_In_Slave_41_Slave_40"}
	ASI_In_Slave_41_Slave_40 AT %I* : USINT;
	{attribute addProperty Name "ASI_In_Slave_43_Slave_42"}
	ASI_In_Slave_43_Slave_42 AT %I* : USINT;
	{attribute addProperty Name "ASI_In_Slave_45_Slave_44"}
	ASI_In_Slave_45_Slave_44 AT %I* : USINT;
	{attribute addProperty Name "ASI_In_Slave_47_Slave_46"}
	ASI_In_Slave_47_Slave_46 AT %I* : USINT;
	{attribute addProperty Name "ASI_In_Slave_49_Slave_48"}
	ASI_In_Slave_49_Slave_48 AT %I* : USINT;
	{attribute addProperty Name "ASI_In_Slave_51_Slave_50"}
	ASI_In_Slave_51_Slave_50 AT %I* : USINT;
	{attribute addProperty Name "ASI_In_Slave_53_Slave_52"}
	ASI_In_Slave_53_Slave_52 AT %I* : USINT;
	{attribute addProperty Name "ASI_In_Slave_55_Slave_54"}
	ASI_In_Slave_55_Slave_54 AT %I* : USINT;
	{attribute addProperty Name "ASI_In_Slave_57_Slave_56"}
	ASI_In_Slave_57_Slave_56 AT %I* : USINT;
	{attribute addProperty Name "ASI_In_Slave_59_Slave_58"}
	ASI_In_Slave_59_Slave_58 AT %I* : USINT;
	{attribute addProperty Name "ASI_In_Slave_61_Slave_60"}
	ASI_In_Slave_61_Slave_60 AT %I* : USINT;
	{attribute addProperty Name "ASI_In_Slave_63_Slave_62"}
	ASI_In_Slave_63_Slave_62 AT %I* : USINT;
	{attribute addProperty Name "Control"}
	Control AT %Q* : UINT;
	{attribute addProperty Name "Parameter_Out"}
	Parameter_Out AT %Q* : UDINT;
	{attribute addProperty Name "ASI_Out_Slave_1_Control"}
	ASI_Out_Slave_1_Control AT %Q* : USINT;
	{attribute addProperty Name "ASI_Out_Slave_3_Slave_2"}
	ASI_Out_Slave_3_Slave_2 AT %Q* : USINT;
	{attribute addProperty Name "ASI_Out_Slave_5_Slave_4"}
	ASI_Out_Slave_5_Slave_4 AT %Q* : USINT;
	{attribute addProperty Name "ASI_Out_Slave_7_Slave_6"}
	ASI_Out_Slave_7_Slave_6 AT %Q* : USINT;
	{attribute addProperty Name "ASI_Out_Slave_9_Slave_8"}
	ASI_Out_Slave_9_Slave_8 AT %Q* : USINT;
	{attribute addProperty Name "ASI_Out_Slave_11_Slave_10"}
	ASI_Out_Slave_11_Slave_10 AT %Q* : USINT;
	{attribute addProperty Name "ASI_Out_Slave_13_Slave_12"}
	ASI_Out_Slave_13_Slave_12 AT %Q* : USINT;
	{attribute addProperty Name "ASI_Out_Slave_15_Slave_14"}
	ASI_Out_Slave_15_Slave_14 AT %Q* : USINT;
	{attribute addProperty Name "ASI_Out_Slave_17_Slave_16"}
	ASI_Out_Slave_17_Slave_16 AT %Q* : USINT;
	{attribute addProperty Name "ASI_Out_Slave_19_Slave_18"}
	ASI_Out_Slave_19_Slave_18 AT %Q* : USINT;
	{attribute addProperty Name "ASI_Out_Slave_21_Slave_20"}
	ASI_Out_Slave_21_Slave_20 AT %Q* : USINT;
	{attribute addProperty Name "ASI_Out_Slave_23_Slave_22"}
	ASI_Out_Slave_23_Slave_22 AT %Q* : USINT;
	{attribute addProperty Name "ASI_Out_Slave_25_Slave_24"}
	ASI_Out_Slave_25_Slave_24 AT %Q* : USINT;
	{attribute addProperty Name "ASI_Out_Slave_27_Slave_26"}
	ASI_Out_Slave_27_Slave_26 AT %Q* : USINT;
	{attribute addProperty Name "ASI_Out_Slave_29_Slave_28"}
	ASI_Out_Slave_29_Slave_28 AT %Q* : USINT;
	{attribute addProperty Name "ASI_Out_Slave_31_Slave_30"}
	ASI_Out_Slave_31_Slave_30 AT %Q* : USINT;
	{attribute addProperty Name "ASI_Out_Slave_33_Slave_32"}
	ASI_Out_Slave_33_Slave_32 AT %Q* : USINT;
	{attribute addProperty Name "ASI_Out_Slave_35_Slave_34"}
	ASI_Out_Slave_35_Slave_34 AT %Q* : USINT;
	{attribute addProperty Name "ASI_Out_Slave_37_Slave_36"}
	ASI_Out_Slave_37_Slave_36 AT %Q* : USINT;
	{attribute addProperty Name "ASI_Out_Slave_39_Slave_38"}
	ASI_Out_Slave_39_Slave_38 AT %Q* : USINT;
	{attribute addProperty Name "ASI_Out_Slave_41_Slave_40"}
	ASI_Out_Slave_41_Slave_40 AT %Q* : USINT;
	{attribute addProperty Name "ASI_Out_Slave_43_Slave_42"}
	ASI_Out_Slave_43_Slave_42 AT %Q* : USINT;
	{attribute addProperty Name "ASI_Out_Slave_45_Slave_44"}
	ASI_Out_Slave_45_Slave_44 AT %Q* : USINT;
	{attribute addProperty Name "ASI_Out_Slave_47_Slave_46"}
	ASI_Out_Slave_47_Slave_46 AT %Q* : USINT;
	{attribute addProperty Name "ASI_Out_Slave_49_Slave_48"}
	ASI_Out_Slave_49_Slave_48 AT %Q* : USINT;
	{attribute addProperty Name "ASI_Out_Slave_51_Slave_50"}
	ASI_Out_Slave_51_Slave_50 AT %Q* : USINT;
	{attribute addProperty Name "ASI_Out_Slave_53_Slave_52"}
	ASI_Out_Slave_53_Slave_52 AT %Q* : USINT;
	{attribute addProperty Name "ASI_Out_Slave_55_Slave_54"}
	ASI_Out_Slave_55_Slave_54 AT %Q* : USINT;
	{attribute addProperty Name "ASI_Out_Slave_57_Slave_56"}
	ASI_Out_Slave_57_Slave_56 AT %Q* : USINT;
	{attribute addProperty Name "ASI_Out_Slave_59_Slave_58"}
	ASI_Out_Slave_59_Slave_58 AT %Q* : USINT;
	{attribute addProperty Name "ASI_Out_Slave_61_Slave_60"}
	ASI_Out_Slave_61_Slave_60 AT %Q* : USINT;
	{attribute addProperty Name "ASI_Out_Slave_63_Slave_62"}
	ASI_Out_Slave_63_Slave_62 AT %Q* : USINT;
END_STRUCT
END_TYPE

// ---- DUTs/IO/PDOs/Channel_A42BCA5C.TcDUT
{attribute 'GeneratedUsingTerminal: KL6211-0024'}
{attribute addProperty BoxType "KL6211-0024"}
{attribute addProperty Id "StatusAT %I*UINT0Parameter_InAT %I*UDINT0ASI_In_StatusAT %I*BYTE0ASI_In_Slave_1AT %I*BYTE0ASI_In_Slave_2AT %I*BYTE0ASI_In_Slave_3AT %I*BYTE0ASI_In_Slave_4AT %I*BYTE0ASI_In_Slave_5AT %I*BYTE0ASI_In_Slave_6AT %I*BYTE0ASI_In_Slave_7AT %I*BYTE0ASI_In_Slave_8AT %I*BYTE0ASI_In_Slave_9AT %I*BYTE0ASI_In_Slave_10AT %I*BYTE0ASI_In_Slave_11AT %I*BYTE0ASI_In_Slave_12AT %I*BYTE0ASI_In_Slave_13AT %I*BYTE0ASI_In_Slave_14AT %I*BYTE0ASI_In_Slave_15AT %I*BYTE0ASI_In_Slave_16AT %I*BYTE0ASI_In_Slave_17AT %I*BYTE0ASI_In_Slave_18AT %I*BYTE0ASI_In_Slave_19AT %I*BYTE0ASI_In_Slave_20AT %I*BYTE0ASI_In_Slave_21AT %I*BYTE0ASI_In_Slave_22AT %I*BYTE0ASI_In_Slave_23AT %I*BYTE0ASI_In_Slave_24AT %I*BYTE0ASI_In_Slave_25AT %I*BYTE0ASI_In_Slave_26AT %I*BYTE0ASI_In_Slave_27AT %I*BYTE0ASI_In_Slave_28AT %I*BYTE0ASI_In_Slave_29AT %I*BYTE0ASI_In_Slave_30AT %I*BYTE0ASI_In_Slave_31AT %I*BYTE0ASI_In_Slave_32AT %I*BYTE0ASI_In_Slave_33AT %I*BYTE0ASI_In_Slave_34AT %I*BYTE0ASI_In_Slave_35AT %I*BYTE0ASI_In_Slave_36AT %I*BYTE0ASI_In_Slave_37AT %I*BYTE0ASI_In_Slave_38AT %I*BYTE0ASI_In_Slave_39AT %I*BYTE0ASI_In_Slave_40AT %I*BYTE0ASI_In_Slave_41AT %I*BYTE0ASI_In_Slave_42AT %I*BYTE0ASI_In_Slave_43AT %I*BYTE0ASI_In_Slave_44AT %I*BYTE0ASI_In_Slave_45AT %I*BYTE0ASI_In_Slave_46AT %I*BYTE0ASI_In_Slave_47AT %I*BYTE0ASI_In_Slave_48AT %I*BYTE0ASI_In_Slave_49AT %I*BYTE0ASI_In_Slave_50AT %I*BYTE0ASI_In_Slave_51AT %I*BYTE0ASI_In_Slave_52AT %I*BYTE0ASI_In_Slave_53AT %I*BYTE0ASI_In_Slave_54AT %I*BYTE0ASI_In_Slave_55AT %I*BYTE0ASI_In_Slave_56AT %I*BYTE0ASI_In_Slave_57AT %I*BYTE0ASI_In_Slave_58AT %I*BYTE0ASI_In_Slave_59AT %I*BYTE0ASI_In_Slave_60AT %I*BYTE0ASI_In_Slave_61AT %I*BYTE0ASI_In_Slave_62AT %I*BYTE0ASI_In_Slave_63AT %I*BYTE0ControlAT %Q*UINT0Parameter_OutAT %Q*UDINT0ASI_Out_ControlAT %Q*BYTE0ASI_Out_Slave_1AT %Q*BYTE0ASI_Out_Slave_2AT %Q*BYTE0ASI_Out_Slave_3AT %Q*BYTE0ASI_Out_Slave_4AT %Q*BYTE0ASI_Out_Slave_5AT %Q*BYTE0ASI_Out_Slave_6AT %Q*BYTE0ASI_Out_Slave_7AT %Q*BYTE0ASI_Out_Slave_8AT %Q*BYTE0ASI_Out_Slave_9AT %Q*BYTE0ASI_Out_Slave_10AT %Q*BYTE0ASI_Out_Slave_11AT %Q*BYTE0ASI_Out_Slave_12AT %Q*BYTE0ASI_Out_Slave_13AT %Q*BYTE0ASI_Out_Slave_14AT %Q*BYTE0ASI_Out_Slave_15AT %Q*BYTE0ASI_Out_Slave_16AT %Q*BYTE0ASI_Out_Slave_17AT %Q*BYTE0ASI_Out_Slave_18AT %Q*BYTE0ASI_Out_Slave_19AT %Q*BYTE0ASI_Out_Slave_20AT %Q*BYTE0ASI_Out_Slave_21AT %Q*BYTE0ASI_Out_Slave_22AT %Q*BYTE0ASI_Out_Slave_23AT %Q*BYTE0ASI_Out_Slave_24AT %Q*BYTE0ASI_Out_Slave_25AT %Q*BYTE0ASI_Out_Slave_26AT %Q*BYTE0ASI_Out_Slave_27AT %Q*BYTE0ASI_Out_Slave_28AT %Q*BYTE0ASI_Out_Slave_29AT %Q*BYTE0ASI_Out_Slave_30AT %Q*BYTE0ASI_Out_Slave_31AT %Q*BYTE0ASI_Out_Slave_32AT %Q*BYTE0ASI_Out_Slave_33AT %Q*BYTE0ASI_Out_Slave_34AT %Q*BYTE0ASI_Out_Slave_35AT %Q*BYTE0ASI_Out_Slave_36AT %Q*BYTE0ASI_Out_Slave_37AT %Q*BYTE0ASI_Out_Slave_38AT %Q*BYTE0ASI_Out_Slave_39AT %Q*BYTE0ASI_Out_Slave_40AT %Q*BYTE0ASI_Out_Slave_41AT %Q*BYTE0ASI_Out_Slave_42AT %Q*BYTE0ASI_Out_Slave_43AT %Q*BYTE0ASI_Out_Slave_44AT %Q*BYTE0ASI_Out_Slave_45AT %Q*BYTE0ASI_Out_Slave_46AT %Q*BYTE0ASI_Out_Slave_47AT %Q*BYTE0ASI_Out_Slave_48AT %Q*BYTE0ASI_Out_Slave_49AT %Q*BYTE0ASI_Out_Slave_50AT %Q*BYTE0ASI_Out_Slave_51AT %Q*BYTE0ASI_Out_Slave_52AT %Q*BYTE0ASI_Out_Slave_53AT %Q*BYTE0ASI_Out_Slave_54AT %Q*BYTE0ASI_Out_Slave_55AT %Q*BYTE0ASI_Out_Slave_56AT %Q*BYTE0ASI_Out_Slave_57AT %Q*BYTE0ASI_Out_Slave_58AT %Q*BYTE0ASI_Out_Slave_59AT %Q*BYTE0ASI_Out_Slave_60AT %Q*BYTE0ASI_Out_Slave_61AT %Q*BYTE0ASI_Out_Slave_62AT %Q*BYTE0ASI_Out_Slave_63AT %Q*BYTE0"}
{attribute addProperty CRC "2754333276"}
{attribute addProperty Size "0"}
TYPE Channel_A42BCA5C :
STRUCT
	{attribute addProperty Name "Status"}
	Status AT %I* : UINT;
	{attribute addProperty Name "Parameter_In"}
	Parameter_In AT %I* : UDINT;
	{attribute addProperty Name "ASI_In_Status"}
	ASI_In_Status AT %I* : BYTE;
	{attribute addProperty Name "ASI_In_Slave_1"}
	ASI_In_Slave_1 AT %I* : BYTE;
	{attribute addProperty Name "ASI_In_Slave_2"}
	ASI_In_Slave_2 AT %I* : BYTE;
	{attribute addProperty Name "ASI_In_Slave_3"}
	ASI_In_Slave_3 AT %I* : BYTE;
	{attribute addProperty Name "ASI_In_Slave_4"}
	ASI_In_Slave_4 AT %I* : BYTE;
	{attribute addProperty Name "ASI_In_Slave_5"}
	ASI_In_Slave_5 AT %I* : BYTE;
	{attribute addProperty Name "ASI_In_Slave_6"}
	ASI_In_Slave_6 AT %I* : BYTE;
	{attribute addProperty Name "ASI_In_Slave_7"}
	ASI_In_Slave_7 AT %I* : BYTE;
	{attribute addProperty Name "ASI_In_Slave_8"}
	ASI_In_Slave_8 AT %I* : BYTE;
	{attribute addProperty Name "ASI_In_Slave_9"}
	ASI_In_Slave_9 AT %I* : BYTE;
	{attribute addProperty Name "ASI_In_Slave_10"}
	ASI_In_Slave_10 AT %I* : BYTE;
	{attribute addProperty Name "ASI_In_Slave_11"}
	ASI_In_Slave_11 AT %I* : BYTE;
	{attribute addProperty Name "ASI_In_Slave_12"}
	ASI_In_Slave_12 AT %I* : BYTE;
	{attribute addProperty Name "ASI_In_Slave_13"}
	ASI_In_Slave_13 AT %I* : BYTE;
	{attribute addProperty Name "ASI_In_Slave_14"}
	ASI_In_Slave_14 AT %I* : BYTE;
	{attribute addProperty Name "ASI_In_Slave_15"}
	ASI_In_Slave_15 AT %I* : BYTE;
	{attribute addProperty Name "ASI_In_Slave_16"}
	ASI_In_Slave_16 AT %I* : BYTE;
	{attribute addProperty Name "ASI_In_Slave_17"}
	ASI_In_Slave_17 AT %I* : BYTE;
	{attribute addProperty Name "ASI_In_Slave_18"}
	ASI_In_Slave_18 AT %I* : BYTE;
	{attribute addProperty Name "ASI_In_Slave_19"}
	ASI_In_Slave_19 AT %I* : BYTE;
	{attribute addProperty Name "ASI_In_Slave_20"}
	ASI_In_Slave_20 AT %I* : BYTE;
	{attribute addProperty Name "ASI_In_Slave_21"}
	ASI_In_Slave_21 AT %I* : BYTE;
	{attribute addProperty Name "ASI_In_Slave_22"}
	ASI_In_Slave_22 AT %I* : BYTE;
	{attribute addProperty Name "ASI_In_Slave_23"}
	ASI_In_Slave_23 AT %I* : BYTE;
	{attribute addProperty Name "ASI_In_Slave_24"}
	ASI_In_Slave_24 AT %I* : BYTE;
	{attribute addProperty Name "ASI_In_Slave_25"}
	ASI_In_Slave_25 AT %I* : BYTE;
	{attribute addProperty Name "ASI_In_Slave_26"}
	ASI_In_Slave_26 AT %I* : BYTE;
	{attribute addProperty Name "ASI_In_Slave_27"}
	ASI_In_Slave_27 AT %I* : BYTE;
	{attribute addProperty Name "ASI_In_Slave_28"}
	ASI_In_Slave_28 AT %I* : BYTE;
	{attribute addProperty Name "ASI_In_Slave_29"}
	ASI_In_Slave_29 AT %I* : BYTE;
	{attribute addProperty Name "ASI_In_Slave_30"}
	ASI_In_Slave_30 AT %I* : BYTE;
	{attribute addProperty Name "ASI_In_Slave_31"}
	ASI_In_Slave_31 AT %I* : BYTE;
	{attribute addProperty Name "ASI_In_Slave_32"}
	ASI_In_Slave_32 AT %I* : BYTE;
	{attribute addProperty Name "ASI_In_Slave_33"}
	ASI_In_Slave_33 AT %I* : BYTE;
	{attribute addProperty Name "ASI_In_Slave_34"}
	ASI_In_Slave_34 AT %I* : BYTE;
	{attribute addProperty Name "ASI_In_Slave_35"}
	ASI_In_Slave_35 AT %I* : BYTE;
	{attribute addProperty Name "ASI_In_Slave_36"}
	ASI_In_Slave_36 AT %I* : BYTE;
	{attribute addProperty Name "ASI_In_Slave_37"}
	ASI_In_Slave_37 AT %I* : BYTE;
	{attribute addProperty Name "ASI_In_Slave_38"}
	ASI_In_Slave_38 AT %I* : BYTE;
	{attribute addProperty Name "ASI_In_Slave_39"}
	ASI_In_Slave_39 AT %I* : BYTE;
	{attribute addProperty Name "ASI_In_Slave_40"}
	ASI_In_Slave_40 AT %I* : BYTE;
	{attribute addProperty Name "ASI_In_Slave_41"}
	ASI_In_Slave_41 AT %I* : BYTE;
	{attribute addProperty Name "ASI_In_Slave_42"}
	ASI_In_Slave_42 AT %I* : BYTE;
	{attribute addProperty Name "ASI_In_Slave_43"}
	ASI_In_Slave_43 AT %I* : BYTE;
	{attribute addProperty Name "ASI_In_Slave_44"}
	ASI_In_Slave_44 AT %I* : BYTE;
	{attribute addProperty Name "ASI_In_Slave_45"}
	ASI_In_Slave_45 AT %I* : BYTE;
	{attribute addProperty Name "ASI_In_Slave_46"}
	ASI_In_Slave_46 AT %I* : BYTE;
	{attribute addProperty Name "ASI_In_Slave_47"}
	ASI_In_Slave_47 AT %I* : BYTE;
	{attribute addProperty Name "ASI_In_Slave_48"}
	ASI_In_Slave_48 AT %I* : BYTE;
	{attribute addProperty Name "ASI_In_Slave_49"}
	ASI_In_Slave_49 AT %I* : BYTE;
	{attribute addProperty Name "ASI_In_Slave_50"}
	ASI_In_Slave_50 AT %I* : BYTE;
	{attribute addProperty Name "ASI_In_Slave_51"}
	ASI_In_Slave_51 AT %I* : BYTE;
	{attribute addProperty Name "ASI_In_Slave_52"}
	ASI_In_Slave_52 AT %I* : BYTE;
	{attribute addProperty Name "ASI_In_Slave_53"}
	ASI_In_Slave_53 AT %I* : BYTE;
	{attribute addProperty Name "ASI_In_Slave_54"}
	ASI_In_Slave_54 AT %I* : BYTE;
	{attribute addProperty Name "ASI_In_Slave_55"}
	ASI_In_Slave_55 AT %I* : BYTE;
	{attribute addProperty Name "ASI_In_Slave_56"}
	ASI_In_Slave_56 AT %I* : BYTE;
	{attribute addProperty Name "ASI_In_Slave_57"}
	ASI_In_Slave_57 AT %I* : BYTE;
	{attribute addProperty Name "ASI_In_Slave_58"}
	ASI_In_Slave_58 AT %I* : BYTE;
	{attribute addProperty Name "ASI_In_Slave_59"}
	ASI_In_Slave_59 AT %I* : BYTE;
	{attribute addProperty Name "ASI_In_Slave_60"}
	ASI_In_Slave_60 AT %I* : BYTE;
	{attribute addProperty Name "ASI_In_Slave_61"}
	ASI_In_Slave_61 AT %I* : BYTE;
	{attribute addProperty Name "ASI_In_Slave_62"}
	ASI_In_Slave_62 AT %I* : BYTE;
	{attribute addProperty Name "ASI_In_Slave_63"}
	ASI_In_Slave_63 AT %I* : BYTE;
	{attribute addProperty Name "Control"}
	Control AT %Q* : UINT;
	{attribute addProperty Name "Parameter_Out"}
	Parameter_Out AT %Q* : UDINT;
	{attribute addProperty Name "ASI_Out_Control"}
	ASI_Out_Control AT %Q* : BYTE;
	{attribute addProperty Name "ASI_Out_Slave_1"}
	ASI_Out_Slave_1 AT %Q* : BYTE;
	{attribute addProperty Name "ASI_Out_Slave_2"}
	ASI_Out_Slave_2 AT %Q* : BYTE;
	{attribute addProperty Name "ASI_Out_Slave_3"}
	ASI_Out_Slave_3 AT %Q* : BYTE;
	{attribute addProperty Name "ASI_Out_Slave_4"}
	ASI_Out_Slave_4 AT %Q* : BYTE;
	{attribute addProperty Name "ASI_Out_Slave_5"}
	ASI_Out_Slave_5 AT %Q* : BYTE;
	{attribute addProperty Name "ASI_Out_Slave_6"}
	ASI_Out_Slave_6 AT %Q* : BYTE;
	{attribute addProperty Name "ASI_Out_Slave_7"}
	ASI_Out_Slave_7 AT %Q* : BYTE;
	{attribute addProperty Name "ASI_Out_Slave_8"}
	ASI_Out_Slave_8 AT %Q* : BYTE;
	{attribute addProperty Name "ASI_Out_Slave_9"}
	ASI_Out_Slave_9 AT %Q* : BYTE;
	{attribute addProperty Name "ASI_Out_Slave_10"}
	ASI_Out_Slave_10 AT %Q* : BYTE;
	{attribute addProperty Name "ASI_Out_Slave_11"}
	ASI_Out_Slave_11 AT %Q* : BYTE;
	{attribute addProperty Name "ASI_Out_Slave_12"}
	ASI_Out_Slave_12 AT %Q* : BYTE;
	{attribute addProperty Name "ASI_Out_Slave_13"}
	ASI_Out_Slave_13 AT %Q* : BYTE;
	{attribute addProperty Name "ASI_Out_Slave_14"}
	ASI_Out_Slave_14 AT %Q* : BYTE;
	{attribute addProperty Name "ASI_Out_Slave_15"}
	ASI_Out_Slave_15 AT %Q* : BYTE;
	{attribute addProperty Name "ASI_Out_Slave_16"}
	ASI_Out_Slave_16 AT %Q* : BYTE;
	{attribute addProperty Name "ASI_Out_Slave_17"}
	ASI_Out_Slave_17 AT %Q* : BYTE;
	{attribute addProperty Name "ASI_Out_Slave_18"}
	ASI_Out_Slave_18 AT %Q* : BYTE;
	{attribute addProperty Name "ASI_Out_Slave_19"}
	ASI_Out_Slave_19 AT %Q* : BYTE;
	{attribute addProperty Name "ASI_Out_Slave_20"}
	ASI_Out_Slave_20 AT %Q* : BYTE;
	{attribute addProperty Name "ASI_Out_Slave_21"}
	ASI_Out_Slave_21 AT %Q* : BYTE;
	{attribute addProperty Name "ASI_Out_Slave_22"}
	ASI_Out_Slave_22 AT %Q* : BYTE;
	{attribute addProperty Name "ASI_Out_Slave_23"}
	ASI_Out_Slave_23 AT %Q* : BYTE;
	{attribute addProperty Name "ASI_Out_Slave_24"}
	ASI_Out_Slave_24 AT %Q* : BYTE;
	{attribute addProperty Name "ASI_Out_Slave_25"}
	ASI_Out_Slave_25 AT %Q* : BYTE;
	{attribute addProperty Name "ASI_Out_Slave_26"}
	ASI_Out_Slave_26 AT %Q* : BYTE;
	{attribute addProperty Name "ASI_Out_Slave_27"}
	ASI_Out_Slave_27 AT %Q* : BYTE;
	{attribute addProperty Name "ASI_Out_Slave_28"}
	ASI_Out_Slave_28 AT %Q* : BYTE;
	{attribute addProperty Name "ASI_Out_Slave_29"}
	ASI_Out_Slave_29 AT %Q* : BYTE;
	{attribute addProperty Name "ASI_Out_Slave_30"}
	ASI_Out_Slave_30 AT %Q* : BYTE;
	{attribute addProperty Name "ASI_Out_Slave_31"}
	ASI_Out_Slave_31 AT %Q* : BYTE;
	{attribute addProperty Name "ASI_Out_Slave_32"}
	ASI_Out_Slave_32 AT %Q* : BYTE;
	{attribute addProperty Name "ASI_Out_Slave_33"}
	ASI_Out_Slave_33 AT %Q* : BYTE;
	{attribute addProperty Name "ASI_Out_Slave_34"}
	ASI_Out_Slave_34 AT %Q* : BYTE;
	{attribute addProperty Name "ASI_Out_Slave_35"}
	ASI_Out_Slave_35 AT %Q* : BYTE;
	{attribute addProperty Name "ASI_Out_Slave_36"}
	ASI_Out_Slave_36 AT %Q* : BYTE;
	{attribute addProperty Name "ASI_Out_Slave_37"}
	ASI_Out_Slave_37 AT %Q* : BYTE;
	{attribute addProperty Name "ASI_Out_Slave_38"}
	ASI_Out_Slave_38 AT %Q* : BYTE;
	{attribute addProperty Name "ASI_Out_Slave_39"}
	ASI_Out_Slave_39 AT %Q* : BYTE;
	{attribute addProperty Name "ASI_Out_Slave_40"}
	ASI_Out_Slave_40 AT %Q* : BYTE;
	{attribute addProperty Name "ASI_Out_Slave_41"}
	ASI_Out_Slave_41 AT %Q* : BYTE;
	{attribute addProperty Name "ASI_Out_Slave_42"}
	ASI_Out_Slave_42 AT %Q* : BYTE;
	{attribute addProperty Name "ASI_Out_Slave_43"}
	ASI_Out_Slave_43 AT %Q* : BYTE;
	{attribute addProperty Name "ASI_Out_Slave_44"}
	ASI_Out_Slave_44 AT %Q* : BYTE;
	{attribute addProperty Name "ASI_Out_Slave_45"}
	ASI_Out_Slave_45 AT %Q* : BYTE;
	{attribute addProperty Name "ASI_Out_Slave_46"}
	ASI_Out_Slave_46 AT %Q* : BYTE;
	{attribute addProperty Name "ASI_Out_Slave_47"}
	ASI_Out_Slave_47 AT %Q* : BYTE;
	{attribute addProperty Name "ASI_Out_Slave_48"}
	ASI_Out_Slave_48 AT %Q* : BYTE;
	{attribute addProperty Name "ASI_Out_Slave_49"}
	ASI_Out_Slave_49 AT %Q* : BYTE;
	{attribute addProperty Name "ASI_Out_Slave_50"}
	ASI_Out_Slave_50 AT %Q* : BYTE;
	{attribute addProperty Name "ASI_Out_Slave_51"}
	ASI_Out_Slave_51 AT %Q* : BYTE;
	{attribute addProperty Name "ASI_Out_Slave_52"}
	ASI_Out_Slave_52 AT %Q* : BYTE;
	{attribute addProperty Name "ASI_Out_Slave_53"}
	ASI_Out_Slave_53 AT %Q* : BYTE;
	{attribute addProperty Name "ASI_Out_Slave_54"}
	ASI_Out_Slave_54 AT %Q* : BYTE;
	{attribute addProperty Name "ASI_Out_Slave_55"}
	ASI_Out_Slave_55 AT %Q* : BYTE;
	{attribute addProperty Name "ASI_Out_Slave_56"}
	ASI_Out_Slave_56 AT %Q* : BYTE;
	{attribute addProperty Name "ASI_Out_Slave_57"}
	ASI_Out_Slave_57 AT %Q* : BYTE;
	{attribute addProperty Name "ASI_Out_Slave_58"}
	ASI_Out_Slave_58 AT %Q* : BYTE;
	{attribute addProperty Name "ASI_Out_Slave_59"}
	ASI_Out_Slave_59 AT %Q* : BYTE;
	{attribute addProperty Name "ASI_Out_Slave_60"}
	ASI_Out_Slave_60 AT %Q* : BYTE;
	{attribute addProperty Name "ASI_Out_Slave_61"}
	ASI_Out_Slave_61 AT %Q* : BYTE;
	{attribute addProperty Name "ASI_Out_Slave_62"}
	ASI_Out_Slave_62 AT %Q* : BYTE;
	{attribute addProperty Name "ASI_Out_Slave_63"}
	ASI_Out_Slave_63 AT %Q* : BYTE;
END_STRUCT
END_TYPE

// ---- DUTs/IO/PDOs/Channel_08506BCE.TcDUT
{attribute 'GeneratedUsingTerminal: KL6224'}
{attribute addProperty BoxType "KL6224"}
{attribute addProperty Id "StatusAT %I*UINT0Parameter_InAT %I*UDINT0State_Ch1AT %I*USINT0State_Ch2AT %I*USINT0State_Ch3AT %I*USINT0State_Ch4AT %I*USINT0Data_In_0AT %I*USINT0Data_In_1AT %I*USINT0ControlAT %Q*UINT0Parameter_OutAT %Q*UDINT0Data_Out_0AT %Q*USINT0Data_Out_1AT %Q*USINT0Data_Out_2AT %Q*USINT0Data_Out_3AT %Q*USINT0Data_Out_4AT %Q*USINT0Data_Out_5AT %Q*USINT0"}
{attribute addProperty CRC "139488206"}
{attribute addProperty Size "0"}
TYPE Channel_08506BCE :
STRUCT
	{attribute addProperty Name "Status"}
	Status AT %I* : UINT;
	{attribute addProperty Name "Parameter_In"}
	Parameter_In AT %I* : UDINT;
	{attribute addProperty Name "State_Ch1"}
	State_Ch1 AT %I* : USINT;
	{attribute addProperty Name "State_Ch2"}
	State_Ch2 AT %I* : USINT;
	{attribute addProperty Name "State_Ch3"}
	State_Ch3 AT %I* : USINT;
	{attribute addProperty Name "State_Ch4"}
	State_Ch4 AT %I* : USINT;
	{attribute addProperty Name "Data_In_0"}
	Data_In_0 AT %I* : USINT;
	{attribute addProperty Name "Data_In_1"}
	Data_In_1 AT %I* : USINT;
	{attribute addProperty Name "Control"}
	Control AT %Q* : UINT;
	{attribute addProperty Name "Parameter_Out"}
	Parameter_Out AT %Q* : UDINT;
	{attribute addProperty Name "Data_Out_0"}
	Data_Out_0 AT %Q* : USINT;
	{attribute addProperty Name "Data_Out_1"}
	Data_Out_1 AT %Q* : USINT;
	{attribute addProperty Name "Data_Out_2"}
	Data_Out_2 AT %Q* : USINT;
	{attribute addProperty Name "Data_Out_3"}
	Data_Out_3 AT %Q* : USINT;
	{attribute addProperty Name "Data_Out_4"}
	Data_Out_4 AT %Q* : USINT;
	{attribute addProperty Name "Data_Out_5"}
	Data_Out_5 AT %Q* : USINT;
END_STRUCT
END_TYPE

// ---- DUTs/IO/PDOs/Channel_08533804.TcDUT
{attribute 'GeneratedUsingTerminal: KL6224-0001'}
{attribute addProperty BoxType "KL6224-0001"}
{attribute addProperty Id "StatusAT %I*UINT0Parameter_InAT %I*UDINT0State_Ch1AT %I*USINT0State_Ch2AT %I*USINT0State_Ch3AT %I*USINT0State_Ch4AT %I*USINT0Data_In_0AT %I*USINT0Data_In_1AT %I*USINT0Data_In_2AT %I*USINT0Data_In_3AT %I*USINT0Data_In_4AT %I*USINT0Data_In_5AT %I*USINT0Data_In_6AT %I*USINT0Data_In_7AT %I*USINT0Data_In_8AT %I*USINT0Data_In_9AT %I*USINT0Data_In_10AT %I*USINT0Data_In_11AT %I*USINT0Data_In_12AT %I*USINT0Data_In_13AT %I*USINT0ControlAT %Q*UINT0Parameter_OutAT %Q*UDINT0Data_Out_0AT %Q*USINT0Data_Out_1AT %Q*USINT0Data_Out_2AT %Q*USINT0Data_Out_3AT %Q*USINT0Data_Out_4AT %Q*USINT0Data_Out_5AT %Q*USINT0Data_Out_6AT %Q*USINT0Data_Out_7AT %Q*USINT0Data_Out_8AT %Q*USINT0Data_Out_9AT %Q*USINT0Data_Out_10AT %Q*USINT0Data_Out_11AT %Q*USINT0Data_Out_12AT %Q*USINT0Data_Out_13AT %Q*USINT0Data_Out_14AT %Q*USINT0Data_Out_15AT %Q*USINT0Data_Out_16AT %Q*USINT0Data_Out_17AT %Q*USINT0"}
{attribute addProperty CRC "139671556"}
{attribute addProperty Size "0"}
TYPE Channel_08533804 :
STRUCT
	{attribute addProperty Name "Status"}
	Status AT %I* : UINT;
	{attribute addProperty Name "Parameter_In"}
	Parameter_In AT %I* : UDINT;
	{attribute addProperty Name "State_Ch1"}
	State_Ch1 AT %I* : USINT;
	{attribute addProperty Name "State_Ch2"}
	State_Ch2 AT %I* : USINT;
	{attribute addProperty Name "State_Ch3"}
	State_Ch3 AT %I* : USINT;
	{attribute addProperty Name "State_Ch4"}
	State_Ch4 AT %I* : USINT;
	{attribute addProperty Name "Data_In_0"}
	Data_In_0 AT %I* : USINT;
	{attribute addProperty Name "Data_In_1"}
	Data_In_1 AT %I* : USINT;
	{attribute addProperty Name "Data_In_2"}
	Data_In_2 AT %I* : USINT;
	{attribute addProperty Name "Data_In_3"}
	Data_In_3 AT %I* : USINT;
	{attribute addProperty Name "Data_In_4"}
	Data_In_4 AT %I* : USINT;
	{attribute addProperty Name "Data_In_5"}
	Data_In_5 AT %I* : USINT;
	{attribute addProperty Name "Data_In_6"}
	Data_In_6 AT %I* : USINT;
	{attribute addProperty Name "Data_In_7"}
	Data_In_7 AT %I* : USINT;
	{attribute addProperty Name "Data_In_8"}
	Data_In_8 AT %I* : USINT;
	{attribute addProperty Name "Data_In_9"}
	Data_In_9 AT %I* : USINT;
	{attribute addProperty Name "Data_In_10"}
	Data_In_10 AT %I* : USINT;
	{attribute addProperty Name "Data_In_11"}
	Data_In_11 AT %I* : USINT;
	{attribute addProperty Name "Data_In_12"}
	Data_In_12 AT %I* : USINT;
	{attribute addProperty Name "Data_In_13"}
	Data_In_13 AT %I* : USINT;
	{attribute addProperty Name "Control"}
	Control AT %Q* : UINT;
	{attribute addProperty Name "Parameter_Out"}
	Parameter_Out AT %Q* : UDINT;
	{attribute addProperty Name "Data_Out_0"}
	Data_Out_0 AT %Q* : USINT;
	{attribute addProperty Name "Data_Out_1"}
	Data_Out_1 AT %Q* : USINT;
	{attribute addProperty Name "Data_Out_2"}
	Data_Out_2 AT %Q* : USINT;
	{attribute addProperty Name "Data_Out_3"}
	Data_Out_3 AT %Q* : USINT;
	{attribute addProperty Name "Data_Out_4"}
	Data_Out_4 AT %Q* : USINT;
	{attribute addProperty Name "Data_Out_5"}
	Data_Out_5 AT %Q* : USINT;
	{attribute addProperty Name "Data_Out_6"}
	Data_Out_6 AT %Q* : USINT;
	{attribute addProperty Name "Data_Out_7"}
	Data_Out_7 AT %Q* : USINT;
	{attribute addProperty Name "Data_Out_8"}
	Data_Out_8 AT %Q* : USINT;
	{attribute addProperty Name "Data_Out_9"}
	Data_Out_9 AT %Q* : USINT;
	{attribute addProperty Name "Data_Out_10"}
	Data_Out_10 AT %Q* : USINT;
	{attribute addProperty Name "Data_Out_11"}
	Data_Out_11 AT %Q* : USINT;
	{attribute addProperty Name "Data_Out_12"}
	Data_Out_12 AT %Q* : USINT;
	{attribute addProperty Name "Data_Out_13"}
	Data_Out_13 AT %Q* : USINT;
	{attribute addProperty Name "Data_Out_14"}
	Data_Out_14 AT %Q* : USINT;
	{attribute addProperty Name "Data_Out_15"}
	Data_Out_15 AT %Q* : USINT;
	{attribute addProperty Name "Data_Out_16"}
	Data_Out_16 AT %Q* : USINT;
	{attribute addProperty Name "Data_Out_17"}
	Data_Out_17 AT %Q* : USINT;
END_STRUCT
END_TYPE

